// TIA Portal V17 export
// export: Created 2025-03-07T09:16:38.8278492Z, ExportSetting WithDefaults, DisplayName Totally Integrated Automation Portal, DisplayVersion V17 Update 8, DisplayName TIA Portal Openness, DisplayVersion V17 Update 8, DisplayName TIA Portal Version Control Interface, DisplayVersion V17, DisplayName SINAMICS Startdrive Advanced, DisplayVersion V17 SP2, DisplayName SINAMICS Startdrive G110M, G120, G120C, G120D, G120P, G115D, DisplayVersion V17 SP2, DisplayName SINAMICS Startdrive G130, G150, S120, S150, SINAMICS MV, S210, DisplayVersion V17 SP2, DisplayName STEP 7 Professional, DisplayVersion V17 Update 8, DisplayName SINUMERIK ONE STEP 7 Toolbox, DisplayVersion V17 Update 12, DisplayName SINUMERIK 840D sl STEP 7 Toolbox, DisplayVersion V17 Update 12, DisplayName STEP 7 Safety, DisplayVersion V17 Update 6, DisplayName WinCC Advanced, DisplayVersion V17 Update 8
FUNCTION "FC2410_PLC_CNC_SIGNALS" : Void   // FC2410, LAD
TITLE = NCK Inputs
{ S7_Optimized_Access := 'FALSE' }
AUTHOR : ETXETAR
VERSION : 1.0
// stored: AutoNumber false, IsIECCheckEnabled false, SetENOAutomatically false, UDAEnableTagReadback false
   VAR_TEMP
      Error : Bool;   // Error
      ErrorCode : Int;   // ErrorCode
   END_VAR
   VAR CONSTANT
      WRITE : Byte := 16#4;
   END_VAR
BEGIN

REGION Network 1: PLC NC SIGNALS 1-8
   // SIGNAL1 --> SEMIAUTO MODE
   // SIGNAL2 --> DRY CYCLE
   // SIGNAL3 --> RUN OUT
   // SIGNAL4 --> BA3
   // SIGNAL5 --> MANUAL LOAD 
   // SIGNAL6 --> GANTRY ROBOT TEST
   // SIGNAL7 --> ROBOT DRY CYCLE
   // SIGNAL8 --> SPARE
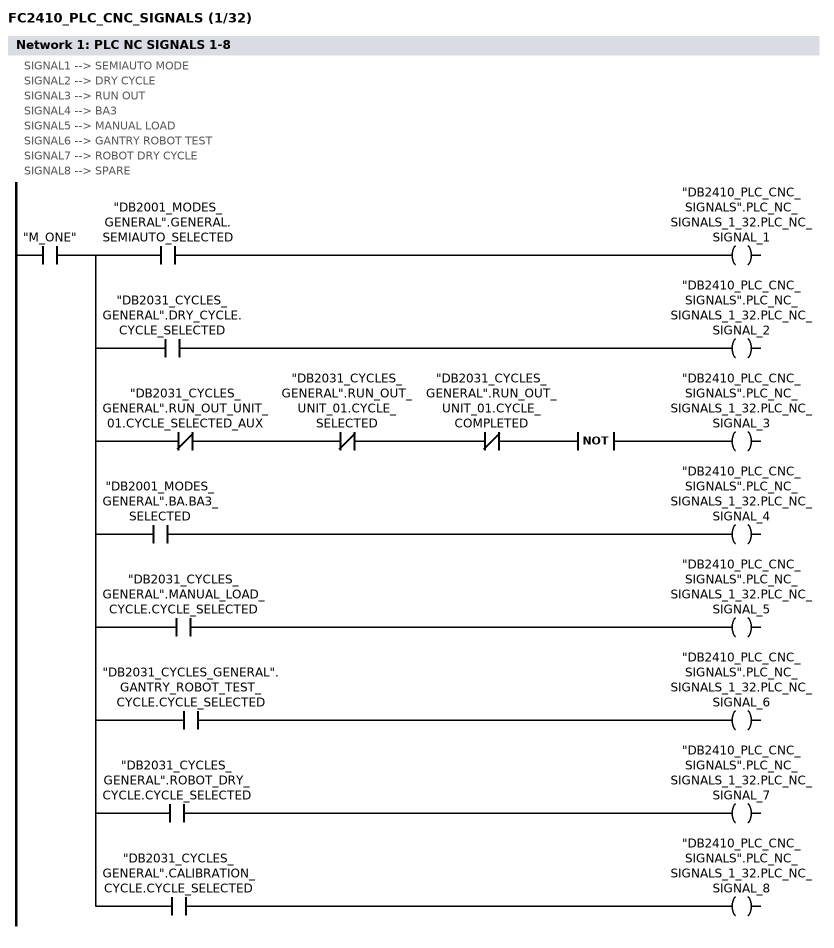
   RUNG wire#powerrail
      Contact( "M_ONE" )
      wire#w1
      Contact( "DB2001_MODES_GENERAL".GENERAL.SEMIAUTO_SELECTED )
      Coil( "DB2410_PLC_CNC_SIGNALS".PLC_NC_SIGNALS_1_32.PLC_NC_SIGNAL_1 )
   END_RUNG
   RUNG wire#w1
      Contact( "DB2031_CYCLES_GENERAL".DRY_CYCLE.CYCLE_SELECTED )
      Coil( "DB2410_PLC_CNC_SIGNALS".PLC_NC_SIGNALS_1_32.PLC_NC_SIGNAL_2 )
   END_RUNG
   RUNG wire#w1
      I_Contact( "DB2031_CYCLES_GENERAL".RUN_OUT_UNIT_01.CYCLE_SELECTED_AUX )
      I_Contact( "DB2031_CYCLES_GENERAL".RUN_OUT_UNIT_01.CYCLE_SELECTED )
      I_Contact( "DB2031_CYCLES_GENERAL".RUN_OUT_UNIT_01.CYCLE_COMPLETED )
      Not()
      Coil( "DB2410_PLC_CNC_SIGNALS".PLC_NC_SIGNALS_1_32.PLC_NC_SIGNAL_3 )
   END_RUNG
   RUNG wire#w1
      Contact( "DB2001_MODES_GENERAL".BA.BA3_SELECTED )
      Coil( "DB2410_PLC_CNC_SIGNALS".PLC_NC_SIGNALS_1_32.PLC_NC_SIGNAL_4 )
   END_RUNG
   RUNG wire#w1
      Contact( "DB2031_CYCLES_GENERAL".MANUAL_LOAD_CYCLE.CYCLE_SELECTED )
      Coil( "DB2410_PLC_CNC_SIGNALS".PLC_NC_SIGNALS_1_32.PLC_NC_SIGNAL_5 )
   END_RUNG
   RUNG wire#w1
      Contact( "DB2031_CYCLES_GENERAL".GANTRY_ROBOT_TEST_CYCLE.CYCLE_SELECTED )
      Coil( "DB2410_PLC_CNC_SIGNALS".PLC_NC_SIGNALS_1_32.PLC_NC_SIGNAL_6 )
   END_RUNG
   RUNG wire#w1
      Contact( "DB2031_CYCLES_GENERAL".ROBOT_DRY_CYCLE.CYCLE_SELECTED )
      Coil( "DB2410_PLC_CNC_SIGNALS".PLC_NC_SIGNALS_1_32.PLC_NC_SIGNAL_7 )
   END_RUNG
   RUNG wire#w1
      Contact( "DB2031_CYCLES_GENERAL".CALIBRATION_CYCLE.CYCLE_SELECTED )
      Coil( "DB2410_PLC_CNC_SIGNALS".PLC_NC_SIGNALS_1_32.PLC_NC_SIGNAL_8 )
   END_RUNG
   // the same network as SCL:
   "DB2410_PLC_CNC_SIGNALS".PLC_NC_SIGNALS_1_32.PLC_NC_SIGNAL_1 := "M_ONE" AND "DB2001_MODES_GENERAL".GENERAL.SEMIAUTO_SELECTED;
   "DB2410_PLC_CNC_SIGNALS".PLC_NC_SIGNALS_1_32.PLC_NC_SIGNAL_2 := "M_ONE" AND "DB2031_CYCLES_GENERAL".DRY_CYCLE.CYCLE_SELECTED;
   "DB2410_PLC_CNC_SIGNALS".PLC_NC_SIGNALS_1_32.PLC_NC_SIGNAL_3 := NOT ("M_ONE" AND NOT "DB2031_CYCLES_GENERAL".RUN_OUT_UNIT_01.CYCLE_SELECTED_AUX AND NOT "DB2031_CYCLES_GENERAL".RUN_OUT_UNIT_01.CYCLE_SELECTED AND NOT "DB2031_CYCLES_GENERAL".RUN_OUT_UNIT_01.CYCLE_COMPLETED);
   "DB2410_PLC_CNC_SIGNALS".PLC_NC_SIGNALS_1_32.PLC_NC_SIGNAL_4 := "M_ONE" AND "DB2001_MODES_GENERAL".BA.BA3_SELECTED;
   "DB2410_PLC_CNC_SIGNALS".PLC_NC_SIGNALS_1_32.PLC_NC_SIGNAL_5 := "M_ONE" AND "DB2031_CYCLES_GENERAL".MANUAL_LOAD_CYCLE.CYCLE_SELECTED;
   "DB2410_PLC_CNC_SIGNALS".PLC_NC_SIGNALS_1_32.PLC_NC_SIGNAL_6 := "M_ONE" AND "DB2031_CYCLES_GENERAL".GANTRY_ROBOT_TEST_CYCLE.CYCLE_SELECTED;
   "DB2410_PLC_CNC_SIGNALS".PLC_NC_SIGNALS_1_32.PLC_NC_SIGNAL_7 := "M_ONE" AND "DB2031_CYCLES_GENERAL".ROBOT_DRY_CYCLE.CYCLE_SELECTED;
   "DB2410_PLC_CNC_SIGNALS".PLC_NC_SIGNALS_1_32.PLC_NC_SIGNAL_8 := "M_ONE" AND "DB2031_CYCLES_GENERAL".CALIBRATION_CYCLE.CYCLE_SELECTED;
END_REGION

REGION Network 2: PLC NC SIGNALS 9-16
   // SIGNAL9 --> SPARE
   // SIGNAL10 --> SPARE
   // SIGNAL11 --> SPARE
   // SIGNAL12 --> SPARE
   // SIGNAL13 --> SPARE
   // SIGNAL14 --> SPARE
   // SIGNAL15 --> SPARE
   // SIGNAL16 --> SPARE
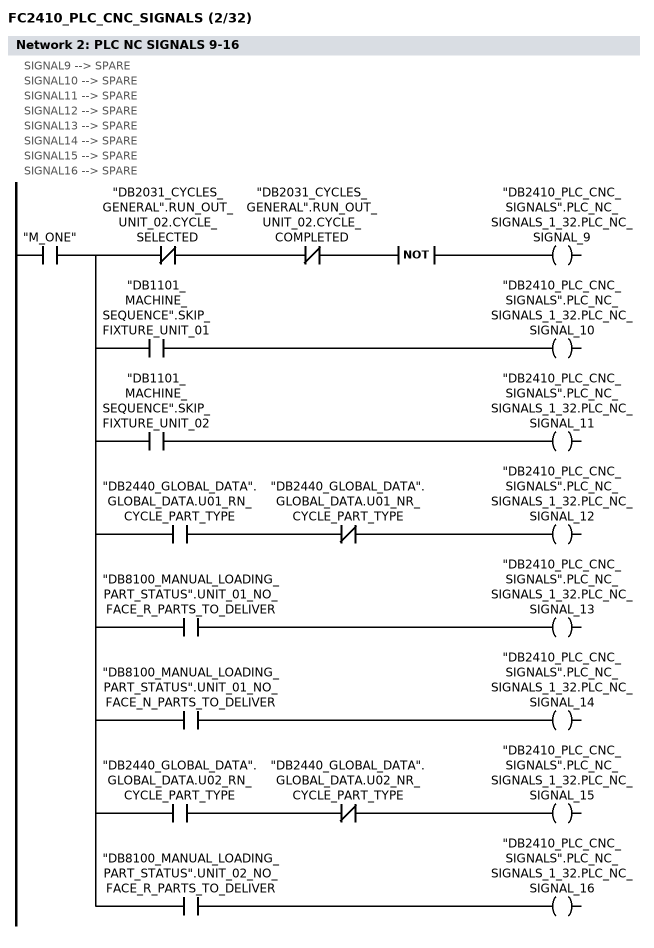
   RUNG wire#powerrail
      Contact( "M_ONE" )
      wire#w1
      I_Contact( "DB2031_CYCLES_GENERAL".RUN_OUT_UNIT_02.CYCLE_SELECTED )
      I_Contact( "DB2031_CYCLES_GENERAL".RUN_OUT_UNIT_02.CYCLE_COMPLETED )
      Not()
      Coil( "DB2410_PLC_CNC_SIGNALS".PLC_NC_SIGNALS_1_32.PLC_NC_SIGNAL_9 )
   END_RUNG
   RUNG wire#w1
      Contact( "DB1101_MACHINE_SEQUENCE".SKIP_FIXTURE_UNIT_01 )
      Coil( "DB2410_PLC_CNC_SIGNALS".PLC_NC_SIGNALS_1_32.PLC_NC_SIGNAL_10 )
   END_RUNG
   RUNG wire#w1
      Contact( "DB1101_MACHINE_SEQUENCE".SKIP_FIXTURE_UNIT_02 )
      Coil( "DB2410_PLC_CNC_SIGNALS".PLC_NC_SIGNALS_1_32.PLC_NC_SIGNAL_11 )
   END_RUNG
   RUNG wire#w1
      Contact( "DB2440_GLOBAL_DATA".GLOBAL_DATA.U01_RN_CYCLE_PART_TYPE )
      I_Contact( "DB2440_GLOBAL_DATA".GLOBAL_DATA.U01_NR_CYCLE_PART_TYPE )
      Coil( "DB2410_PLC_CNC_SIGNALS".PLC_NC_SIGNALS_1_32.PLC_NC_SIGNAL_12 )
   END_RUNG
   RUNG wire#w1
      Contact( "DB8100_MANUAL_LOADING_PART_STATUS".UNIT_01_NO_FACE_R_PARTS_TO_DELIVER )
      Coil( "DB2410_PLC_CNC_SIGNALS".PLC_NC_SIGNALS_1_32.PLC_NC_SIGNAL_13 )
   END_RUNG
   RUNG wire#w1
      Contact( "DB8100_MANUAL_LOADING_PART_STATUS".UNIT_01_NO_FACE_N_PARTS_TO_DELIVER )
      Coil( "DB2410_PLC_CNC_SIGNALS".PLC_NC_SIGNALS_1_32.PLC_NC_SIGNAL_14 )
   END_RUNG
   RUNG wire#w1
      Contact( "DB2440_GLOBAL_DATA".GLOBAL_DATA.U02_RN_CYCLE_PART_TYPE )
      I_Contact( "DB2440_GLOBAL_DATA".GLOBAL_DATA.U02_NR_CYCLE_PART_TYPE )
      Coil( "DB2410_PLC_CNC_SIGNALS".PLC_NC_SIGNALS_1_32.PLC_NC_SIGNAL_15 )
   END_RUNG
   RUNG wire#w1
      Contact( "DB8100_MANUAL_LOADING_PART_STATUS".UNIT_02_NO_FACE_R_PARTS_TO_DELIVER )
      Coil( "DB2410_PLC_CNC_SIGNALS".PLC_NC_SIGNALS_1_32.PLC_NC_SIGNAL_16 )
   END_RUNG
   // the same network as SCL:
   "DB2410_PLC_CNC_SIGNALS".PLC_NC_SIGNALS_1_32.PLC_NC_SIGNAL_9 := NOT ("M_ONE" AND NOT "DB2031_CYCLES_GENERAL".RUN_OUT_UNIT_02.CYCLE_SELECTED AND NOT "DB2031_CYCLES_GENERAL".RUN_OUT_UNIT_02.CYCLE_COMPLETED);
   "DB2410_PLC_CNC_SIGNALS".PLC_NC_SIGNALS_1_32.PLC_NC_SIGNAL_10 := "M_ONE" AND "DB1101_MACHINE_SEQUENCE".SKIP_FIXTURE_UNIT_01;
   "DB2410_PLC_CNC_SIGNALS".PLC_NC_SIGNALS_1_32.PLC_NC_SIGNAL_11 := "M_ONE" AND "DB1101_MACHINE_SEQUENCE".SKIP_FIXTURE_UNIT_02;
   "DB2410_PLC_CNC_SIGNALS".PLC_NC_SIGNALS_1_32.PLC_NC_SIGNAL_12 := "M_ONE" AND "DB2440_GLOBAL_DATA".GLOBAL_DATA.U01_RN_CYCLE_PART_TYPE AND NOT "DB2440_GLOBAL_DATA".GLOBAL_DATA.U01_NR_CYCLE_PART_TYPE;
   "DB2410_PLC_CNC_SIGNALS".PLC_NC_SIGNALS_1_32.PLC_NC_SIGNAL_13 := "M_ONE" AND "DB8100_MANUAL_LOADING_PART_STATUS".UNIT_01_NO_FACE_R_PARTS_TO_DELIVER;
   "DB2410_PLC_CNC_SIGNALS".PLC_NC_SIGNALS_1_32.PLC_NC_SIGNAL_14 := "M_ONE" AND "DB8100_MANUAL_LOADING_PART_STATUS".UNIT_01_NO_FACE_N_PARTS_TO_DELIVER;
   "DB2410_PLC_CNC_SIGNALS".PLC_NC_SIGNALS_1_32.PLC_NC_SIGNAL_15 := "M_ONE" AND "DB2440_GLOBAL_DATA".GLOBAL_DATA.U02_RN_CYCLE_PART_TYPE AND NOT "DB2440_GLOBAL_DATA".GLOBAL_DATA.U02_NR_CYCLE_PART_TYPE;
   "DB2410_PLC_CNC_SIGNALS".PLC_NC_SIGNALS_1_32.PLC_NC_SIGNAL_16 := "M_ONE" AND "DB8100_MANUAL_LOADING_PART_STATUS".UNIT_02_NO_FACE_R_PARTS_TO_DELIVER;
END_REGION

REGION Network 3: PLC NC SIGNALS 17-24
   // SIGNAL17 --> STOP END OF CYCLE
   // SIGNAL18 --> SPARE
   // SIGNAL19 --> SPARE
   // SIGNAL20 --> SPARE
   // SIGNAL21 --> SPARE
   // SIGNAL22 --> SPARE
   // SIGNAL23 --> SPARE
   // SIGNAL24 --> SPARE
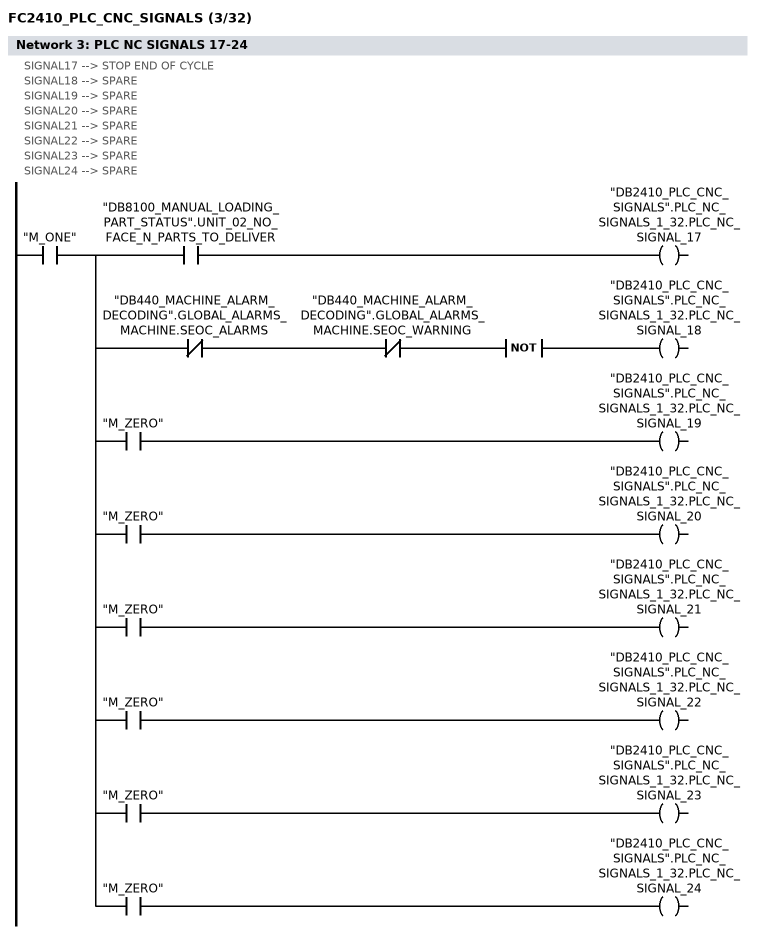
   RUNG wire#powerrail
      Contact( "M_ONE" )
      wire#w1
      Contact( "DB8100_MANUAL_LOADING_PART_STATUS".UNIT_02_NO_FACE_N_PARTS_TO_DELIVER )
      Coil( "DB2410_PLC_CNC_SIGNALS".PLC_NC_SIGNALS_1_32.PLC_NC_SIGNAL_17 )
   END_RUNG
   RUNG wire#w1
      I_Contact( "DB440_MACHINE_ALARM_DECODING".GLOBAL_ALARMS_MACHINE.SEOC_ALARMS )
      I_Contact( "DB440_MACHINE_ALARM_DECODING".GLOBAL_ALARMS_MACHINE.SEOC_WARNING )
      Not()
      Coil( "DB2410_PLC_CNC_SIGNALS".PLC_NC_SIGNALS_1_32.PLC_NC_SIGNAL_18 )
   END_RUNG
   RUNG wire#w1
      Contact( "M_ZERO" )
      Coil( "DB2410_PLC_CNC_SIGNALS".PLC_NC_SIGNALS_1_32.PLC_NC_SIGNAL_19 )
   END_RUNG
   RUNG wire#w1
      Contact( "M_ZERO" )
      Coil( "DB2410_PLC_CNC_SIGNALS".PLC_NC_SIGNALS_1_32.PLC_NC_SIGNAL_20 )
   END_RUNG
   RUNG wire#w1
      Contact( "M_ZERO" )
      Coil( "DB2410_PLC_CNC_SIGNALS".PLC_NC_SIGNALS_1_32.PLC_NC_SIGNAL_21 )
   END_RUNG
   RUNG wire#w1
      Contact( "M_ZERO" )
      Coil( "DB2410_PLC_CNC_SIGNALS".PLC_NC_SIGNALS_1_32.PLC_NC_SIGNAL_22 )
   END_RUNG
   RUNG wire#w1
      Contact( "M_ZERO" )
      Coil( "DB2410_PLC_CNC_SIGNALS".PLC_NC_SIGNALS_1_32.PLC_NC_SIGNAL_23 )
   END_RUNG
   RUNG wire#w1
      Contact( "M_ZERO" )
      Coil( "DB2410_PLC_CNC_SIGNALS".PLC_NC_SIGNALS_1_32.PLC_NC_SIGNAL_24 )
   END_RUNG
   // the same network as SCL:
   "DB2410_PLC_CNC_SIGNALS".PLC_NC_SIGNALS_1_32.PLC_NC_SIGNAL_17 := "M_ONE" AND "DB8100_MANUAL_LOADING_PART_STATUS".UNIT_02_NO_FACE_N_PARTS_TO_DELIVER;
   "DB2410_PLC_CNC_SIGNALS".PLC_NC_SIGNALS_1_32.PLC_NC_SIGNAL_18 := NOT ("M_ONE" AND NOT "DB440_MACHINE_ALARM_DECODING".GLOBAL_ALARMS_MACHINE.SEOC_ALARMS AND NOT "DB440_MACHINE_ALARM_DECODING".GLOBAL_ALARMS_MACHINE.SEOC_WARNING);
   "DB2410_PLC_CNC_SIGNALS".PLC_NC_SIGNALS_1_32.PLC_NC_SIGNAL_19 := "M_ONE" AND "M_ZERO";
   "DB2410_PLC_CNC_SIGNALS".PLC_NC_SIGNALS_1_32.PLC_NC_SIGNAL_20 := "M_ONE" AND "M_ZERO";
   "DB2410_PLC_CNC_SIGNALS".PLC_NC_SIGNALS_1_32.PLC_NC_SIGNAL_21 := "M_ONE" AND "M_ZERO";
   "DB2410_PLC_CNC_SIGNALS".PLC_NC_SIGNALS_1_32.PLC_NC_SIGNAL_22 := "M_ONE" AND "M_ZERO";
   "DB2410_PLC_CNC_SIGNALS".PLC_NC_SIGNALS_1_32.PLC_NC_SIGNAL_23 := "M_ONE" AND "M_ZERO";
   "DB2410_PLC_CNC_SIGNALS".PLC_NC_SIGNALS_1_32.PLC_NC_SIGNAL_24 := "M_ONE" AND "M_ZERO";
END_REGION

REGION Network 4: PLC NC SIGNALS 25-32
   // SIGNAL25 --> CLEAR TO LOAD UNLOAD MACHINE UNIT 01
   // SIGNAL26 --> CLEAR TO LOAD UNLOAD MACHINE UNIT 02
   // SIGNAL27 --> ROBOT OUT OF COLLISION UNIT 01
   // SIGNAL28 --> ROBOT OUT OF COLLISION UNIT 02
   // SIGNAL29 --> SPARE
   // SIGNAL30 --> SPARE
   // SIGNAL31 --> SPARE
   // SIGNAL32 --> SPARE
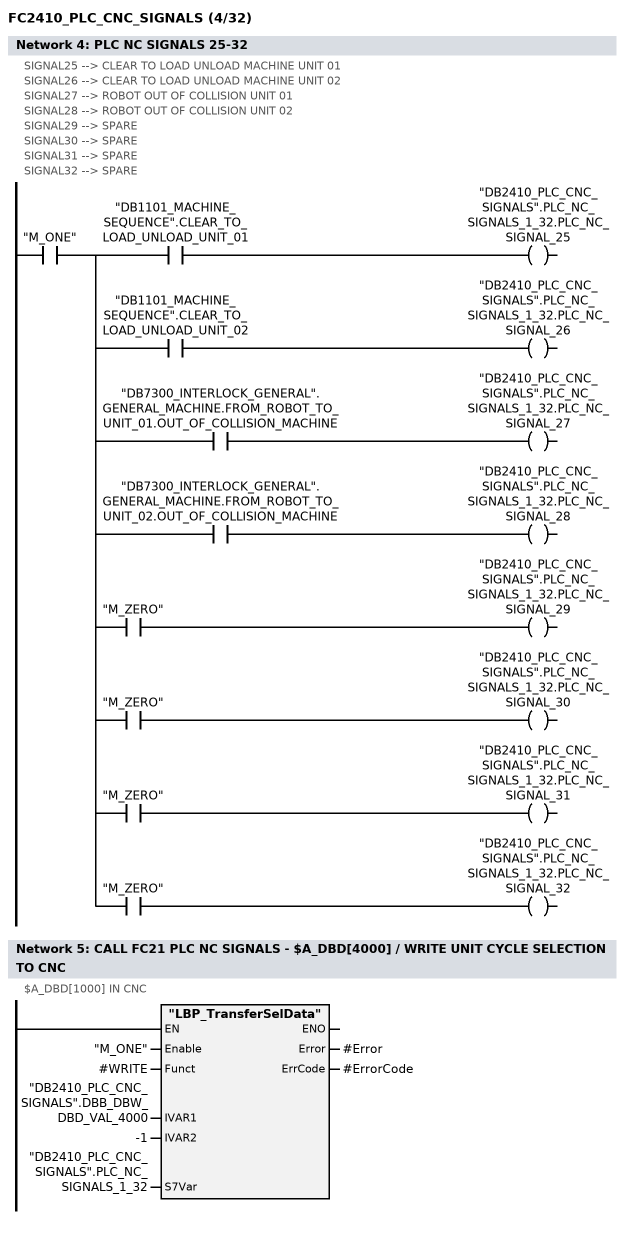
   RUNG wire#powerrail
      Contact( "M_ONE" )
      wire#w1
      Contact( "DB1101_MACHINE_SEQUENCE".CLEAR_TO_LOAD_UNLOAD_UNIT_01 )
      Coil( "DB2410_PLC_CNC_SIGNALS".PLC_NC_SIGNALS_1_32.PLC_NC_SIGNAL_25 )
   END_RUNG
   RUNG wire#w1
      Contact( "DB1101_MACHINE_SEQUENCE".CLEAR_TO_LOAD_UNLOAD_UNIT_02 )
      Coil( "DB2410_PLC_CNC_SIGNALS".PLC_NC_SIGNALS_1_32.PLC_NC_SIGNAL_26 )
   END_RUNG
   RUNG wire#w1
      Contact( "DB7300_INTERLOCK_GENERAL".GENERAL_MACHINE.FROM_ROBOT_TO_UNIT_01.OUT_OF_COLLISION_MACHINE )
      Coil( "DB2410_PLC_CNC_SIGNALS".PLC_NC_SIGNALS_1_32.PLC_NC_SIGNAL_27 )
   END_RUNG
   RUNG wire#w1
      Contact( "DB7300_INTERLOCK_GENERAL".GENERAL_MACHINE.FROM_ROBOT_TO_UNIT_02.OUT_OF_COLLISION_MACHINE )
      Coil( "DB2410_PLC_CNC_SIGNALS".PLC_NC_SIGNALS_1_32.PLC_NC_SIGNAL_28 )
   END_RUNG
   RUNG wire#w1
      Contact( "M_ZERO" )
      Coil( "DB2410_PLC_CNC_SIGNALS".PLC_NC_SIGNALS_1_32.PLC_NC_SIGNAL_29 )
   END_RUNG
   RUNG wire#w1
      Contact( "M_ZERO" )
      Coil( "DB2410_PLC_CNC_SIGNALS".PLC_NC_SIGNALS_1_32.PLC_NC_SIGNAL_30 )
   END_RUNG
   RUNG wire#w1
      Contact( "M_ZERO" )
      Coil( "DB2410_PLC_CNC_SIGNALS".PLC_NC_SIGNALS_1_32.PLC_NC_SIGNAL_31 )
   END_RUNG
   RUNG wire#w1
      Contact( "M_ZERO" )
      Coil( "DB2410_PLC_CNC_SIGNALS".PLC_NC_SIGNALS_1_32.PLC_NC_SIGNAL_32 )
   END_RUNG
   // the same network as SCL:
   "DB2410_PLC_CNC_SIGNALS".PLC_NC_SIGNALS_1_32.PLC_NC_SIGNAL_25 := "M_ONE" AND "DB1101_MACHINE_SEQUENCE".CLEAR_TO_LOAD_UNLOAD_UNIT_01;
   "DB2410_PLC_CNC_SIGNALS".PLC_NC_SIGNALS_1_32.PLC_NC_SIGNAL_26 := "M_ONE" AND "DB1101_MACHINE_SEQUENCE".CLEAR_TO_LOAD_UNLOAD_UNIT_02;
   "DB2410_PLC_CNC_SIGNALS".PLC_NC_SIGNALS_1_32.PLC_NC_SIGNAL_27 := "M_ONE" AND "DB7300_INTERLOCK_GENERAL".GENERAL_MACHINE.FROM_ROBOT_TO_UNIT_01.OUT_OF_COLLISION_MACHINE;
   "DB2410_PLC_CNC_SIGNALS".PLC_NC_SIGNALS_1_32.PLC_NC_SIGNAL_28 := "M_ONE" AND "DB7300_INTERLOCK_GENERAL".GENERAL_MACHINE.FROM_ROBOT_TO_UNIT_02.OUT_OF_COLLISION_MACHINE;
   "DB2410_PLC_CNC_SIGNALS".PLC_NC_SIGNALS_1_32.PLC_NC_SIGNAL_29 := "M_ONE" AND "M_ZERO";
   "DB2410_PLC_CNC_SIGNALS".PLC_NC_SIGNALS_1_32.PLC_NC_SIGNAL_30 := "M_ONE" AND "M_ZERO";
   "DB2410_PLC_CNC_SIGNALS".PLC_NC_SIGNALS_1_32.PLC_NC_SIGNAL_31 := "M_ONE" AND "M_ZERO";
   "DB2410_PLC_CNC_SIGNALS".PLC_NC_SIGNALS_1_32.PLC_NC_SIGNAL_32 := "M_ONE" AND "M_ZERO";
END_REGION

REGION Network 5: CALL FC21 PLC NC SIGNALS - $A_DBD[4000] / WRITE UNIT CYCLE SELECTION TO CNC
   // $A_DBD[1000] IN CNC
   RUNG wire#powerrail
      "LBP_TransferSelData"(Enable := "M_ONE", Funct := #WRITE, IVAR1 := "DB2410_PLC_CNC_SIGNALS".DBB_DBW_DBD_VAL_4000, IVAR2 := -1, S7Var := "DB2410_PLC_CNC_SIGNALS".PLC_NC_SIGNALS_1_32, Error => #Error, ErrCode => #ErrorCode)
   END_RUNG
   // the same network as SCL:
   "LBP_TransferSelData"(Enable := "M_ONE",
                         Funct := #WRITE,
                         IVAR1 := "DB2410_PLC_CNC_SIGNALS".DBB_DBW_DBD_VAL_4000,
                         IVAR2 := -1,
                         S7Var := "DB2410_PLC_CNC_SIGNALS".PLC_NC_SIGNALS_1_32,
                         Error => #Error,
                         ErrCode => #ErrorCode);
END_REGION

REGION Network 6: PLC NC SIGNALS 33-40
   // SIGNAL33 --> TOOL MAZAGINE CHECK HOLDERS 01R
   // SIGNAL34 --> CLEAN TOOL HOLDERS ENABLED 01R
   // SIGNAL35 --> RFID ENABLED 01R
   // SIGNAL36 --> TOOL RFID TAG PRESENT 01R
   // SIGNAL37 --> TOOL CLAMPING DIFFERENCE ALARM 01R
   // SIGNAL38 --> PROBE ENABLED 01R
   // SIGNAL39 --> SPARE
   // SIGNAL40 --> SPARE
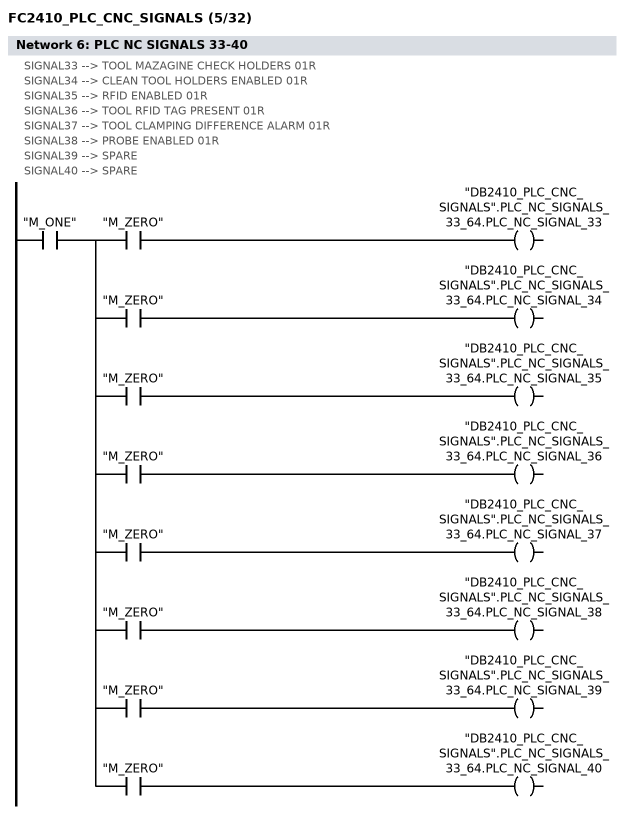
   RUNG wire#powerrail
      Contact( "M_ONE" )
      wire#w1
      Contact( "M_ZERO" )
      Coil( "DB2410_PLC_CNC_SIGNALS".PLC_NC_SIGNALS_33_64.PLC_NC_SIGNAL_33 )
   END_RUNG
   RUNG wire#w1
      Contact( "M_ZERO" )
      Coil( "DB2410_PLC_CNC_SIGNALS".PLC_NC_SIGNALS_33_64.PLC_NC_SIGNAL_34 )
   END_RUNG
   RUNG wire#w1
      Contact( "M_ZERO" )
      Coil( "DB2410_PLC_CNC_SIGNALS".PLC_NC_SIGNALS_33_64.PLC_NC_SIGNAL_35 )
   END_RUNG
   RUNG wire#w1
      Contact( "M_ZERO" )
      Coil( "DB2410_PLC_CNC_SIGNALS".PLC_NC_SIGNALS_33_64.PLC_NC_SIGNAL_36 )
   END_RUNG
   RUNG wire#w1
      Contact( "M_ZERO" )
      Coil( "DB2410_PLC_CNC_SIGNALS".PLC_NC_SIGNALS_33_64.PLC_NC_SIGNAL_37 )
   END_RUNG
   RUNG wire#w1
      Contact( "M_ZERO" )
      Coil( "DB2410_PLC_CNC_SIGNALS".PLC_NC_SIGNALS_33_64.PLC_NC_SIGNAL_38 )
   END_RUNG
   RUNG wire#w1
      Contact( "M_ZERO" )
      Coil( "DB2410_PLC_CNC_SIGNALS".PLC_NC_SIGNALS_33_64.PLC_NC_SIGNAL_39 )
   END_RUNG
   RUNG wire#w1
      Contact( "M_ZERO" )
      Coil( "DB2410_PLC_CNC_SIGNALS".PLC_NC_SIGNALS_33_64.PLC_NC_SIGNAL_40 )
   END_RUNG
   // the same network as SCL:
   "DB2410_PLC_CNC_SIGNALS".PLC_NC_SIGNALS_33_64.PLC_NC_SIGNAL_33 := "M_ONE" AND "M_ZERO";
   "DB2410_PLC_CNC_SIGNALS".PLC_NC_SIGNALS_33_64.PLC_NC_SIGNAL_34 := "M_ONE" AND "M_ZERO";
   "DB2410_PLC_CNC_SIGNALS".PLC_NC_SIGNALS_33_64.PLC_NC_SIGNAL_35 := "M_ONE" AND "M_ZERO";
   "DB2410_PLC_CNC_SIGNALS".PLC_NC_SIGNALS_33_64.PLC_NC_SIGNAL_36 := "M_ONE" AND "M_ZERO";
   "DB2410_PLC_CNC_SIGNALS".PLC_NC_SIGNALS_33_64.PLC_NC_SIGNAL_37 := "M_ONE" AND "M_ZERO";
   "DB2410_PLC_CNC_SIGNALS".PLC_NC_SIGNALS_33_64.PLC_NC_SIGNAL_38 := "M_ONE" AND "M_ZERO";
   "DB2410_PLC_CNC_SIGNALS".PLC_NC_SIGNALS_33_64.PLC_NC_SIGNAL_39 := "M_ONE" AND "M_ZERO";
   "DB2410_PLC_CNC_SIGNALS".PLC_NC_SIGNALS_33_64.PLC_NC_SIGNAL_40 := "M_ONE" AND "M_ZERO";
END_REGION

REGION Network 7: PLC NC SIGNALS 41-48
   // SIGNAL41 --> SPARE
   // SIGNAL42 --> SPARE
   // SIGNAL43 --> SPARE
   // SIGNAL44 --> SPARE
   // SIGNAL45 --> SPARE
   // SIGNAL46 --> SPARE
   // SIGNAL47 --> SPARE
   // SIGNAL48 --> SPARE
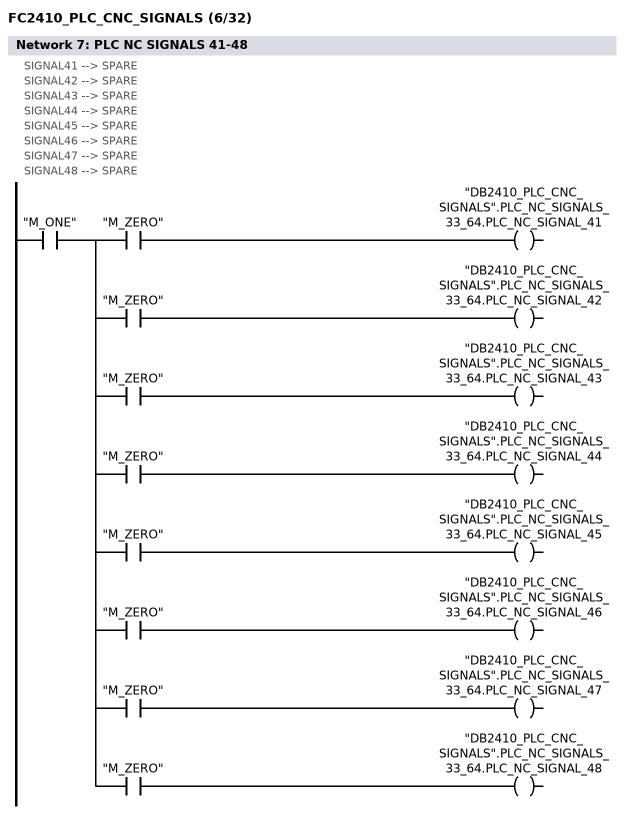
   RUNG wire#powerrail
      Contact( "M_ONE" )
      wire#w1
      Contact( "M_ZERO" )
      Coil( "DB2410_PLC_CNC_SIGNALS".PLC_NC_SIGNALS_33_64.PLC_NC_SIGNAL_41 )
   END_RUNG
   RUNG wire#w1
      Contact( "M_ZERO" )
      Coil( "DB2410_PLC_CNC_SIGNALS".PLC_NC_SIGNALS_33_64.PLC_NC_SIGNAL_42 )
   END_RUNG
   RUNG wire#w1
      Contact( "M_ZERO" )
      Coil( "DB2410_PLC_CNC_SIGNALS".PLC_NC_SIGNALS_33_64.PLC_NC_SIGNAL_43 )
   END_RUNG
   RUNG wire#w1
      Contact( "M_ZERO" )
      Coil( "DB2410_PLC_CNC_SIGNALS".PLC_NC_SIGNALS_33_64.PLC_NC_SIGNAL_44 )
   END_RUNG
   RUNG wire#w1
      Contact( "M_ZERO" )
      Coil( "DB2410_PLC_CNC_SIGNALS".PLC_NC_SIGNALS_33_64.PLC_NC_SIGNAL_45 )
   END_RUNG
   RUNG wire#w1
      Contact( "M_ZERO" )
      Coil( "DB2410_PLC_CNC_SIGNALS".PLC_NC_SIGNALS_33_64.PLC_NC_SIGNAL_46 )
   END_RUNG
   RUNG wire#w1
      Contact( "M_ZERO" )
      Coil( "DB2410_PLC_CNC_SIGNALS".PLC_NC_SIGNALS_33_64.PLC_NC_SIGNAL_47 )
   END_RUNG
   RUNG wire#w1
      Contact( "M_ZERO" )
      Coil( "DB2410_PLC_CNC_SIGNALS".PLC_NC_SIGNALS_33_64.PLC_NC_SIGNAL_48 )
   END_RUNG
   // the same network as SCL:
   "DB2410_PLC_CNC_SIGNALS".PLC_NC_SIGNALS_33_64.PLC_NC_SIGNAL_41 := "M_ONE" AND "M_ZERO";
   "DB2410_PLC_CNC_SIGNALS".PLC_NC_SIGNALS_33_64.PLC_NC_SIGNAL_42 := "M_ONE" AND "M_ZERO";
   "DB2410_PLC_CNC_SIGNALS".PLC_NC_SIGNALS_33_64.PLC_NC_SIGNAL_43 := "M_ONE" AND "M_ZERO";
   "DB2410_PLC_CNC_SIGNALS".PLC_NC_SIGNALS_33_64.PLC_NC_SIGNAL_44 := "M_ONE" AND "M_ZERO";
   "DB2410_PLC_CNC_SIGNALS".PLC_NC_SIGNALS_33_64.PLC_NC_SIGNAL_45 := "M_ONE" AND "M_ZERO";
   "DB2410_PLC_CNC_SIGNALS".PLC_NC_SIGNALS_33_64.PLC_NC_SIGNAL_46 := "M_ONE" AND "M_ZERO";
   "DB2410_PLC_CNC_SIGNALS".PLC_NC_SIGNALS_33_64.PLC_NC_SIGNAL_47 := "M_ONE" AND "M_ZERO";
   "DB2410_PLC_CNC_SIGNALS".PLC_NC_SIGNALS_33_64.PLC_NC_SIGNAL_48 := "M_ONE" AND "M_ZERO";
END_REGION

REGION Network 8: PLC NC SIGNALS 49-56
   // SIGNAL49 --> TOOL MAZAGINE CHECK HOLDERS 01L
   // SIGNAL50 --> CLEAN TOOL HOLDERS ENABLED 01L
   // SIGNAL51 --> RFID ENABLED 01L
   // SIGNAL52 --> TOOL RFID TAG PRESENT 01L
   // SIGNAL53 --> TOOL CLAMPING DIFFERENCE ALARM 01L
   // SIGNAL54 --> PROBE ENABLED 01L
   // SIGNAL55 --> SPARE
   // SIGNAL56 --> SPARE
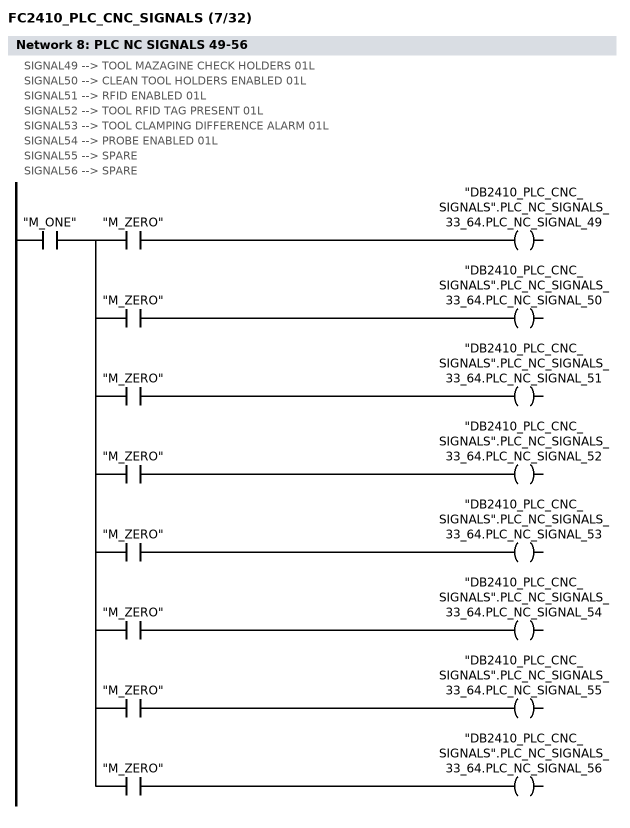
   RUNG wire#powerrail
      Contact( "M_ONE" )
      wire#w1
      Contact( "M_ZERO" )
      Coil( "DB2410_PLC_CNC_SIGNALS".PLC_NC_SIGNALS_33_64.PLC_NC_SIGNAL_49 )
   END_RUNG
   RUNG wire#w1
      Contact( "M_ZERO" )
      Coil( "DB2410_PLC_CNC_SIGNALS".PLC_NC_SIGNALS_33_64.PLC_NC_SIGNAL_50 )
   END_RUNG
   RUNG wire#w1
      Contact( "M_ZERO" )
      Coil( "DB2410_PLC_CNC_SIGNALS".PLC_NC_SIGNALS_33_64.PLC_NC_SIGNAL_51 )
   END_RUNG
   RUNG wire#w1
      Contact( "M_ZERO" )
      Coil( "DB2410_PLC_CNC_SIGNALS".PLC_NC_SIGNALS_33_64.PLC_NC_SIGNAL_52 )
   END_RUNG
   RUNG wire#w1
      Contact( "M_ZERO" )
      Coil( "DB2410_PLC_CNC_SIGNALS".PLC_NC_SIGNALS_33_64.PLC_NC_SIGNAL_53 )
   END_RUNG
   RUNG wire#w1
      Contact( "M_ZERO" )
      Coil( "DB2410_PLC_CNC_SIGNALS".PLC_NC_SIGNALS_33_64.PLC_NC_SIGNAL_54 )
   END_RUNG
   RUNG wire#w1
      Contact( "M_ZERO" )
      Coil( "DB2410_PLC_CNC_SIGNALS".PLC_NC_SIGNALS_33_64.PLC_NC_SIGNAL_55 )
   END_RUNG
   RUNG wire#w1
      Contact( "M_ZERO" )
      Coil( "DB2410_PLC_CNC_SIGNALS".PLC_NC_SIGNALS_33_64.PLC_NC_SIGNAL_56 )
   END_RUNG
   // the same network as SCL:
   "DB2410_PLC_CNC_SIGNALS".PLC_NC_SIGNALS_33_64.PLC_NC_SIGNAL_49 := "M_ONE" AND "M_ZERO";
   "DB2410_PLC_CNC_SIGNALS".PLC_NC_SIGNALS_33_64.PLC_NC_SIGNAL_50 := "M_ONE" AND "M_ZERO";
   "DB2410_PLC_CNC_SIGNALS".PLC_NC_SIGNALS_33_64.PLC_NC_SIGNAL_51 := "M_ONE" AND "M_ZERO";
   "DB2410_PLC_CNC_SIGNALS".PLC_NC_SIGNALS_33_64.PLC_NC_SIGNAL_52 := "M_ONE" AND "M_ZERO";
   "DB2410_PLC_CNC_SIGNALS".PLC_NC_SIGNALS_33_64.PLC_NC_SIGNAL_53 := "M_ONE" AND "M_ZERO";
   "DB2410_PLC_CNC_SIGNALS".PLC_NC_SIGNALS_33_64.PLC_NC_SIGNAL_54 := "M_ONE" AND "M_ZERO";
   "DB2410_PLC_CNC_SIGNALS".PLC_NC_SIGNALS_33_64.PLC_NC_SIGNAL_55 := "M_ONE" AND "M_ZERO";
   "DB2410_PLC_CNC_SIGNALS".PLC_NC_SIGNALS_33_64.PLC_NC_SIGNAL_56 := "M_ONE" AND "M_ZERO";
END_REGION

REGION Network 9: PLC NC SIGNALS 57-64
   // SIGNAL57 --> SPARE
   // SIGNAL58 --> SPARE
   // SIGNAL59 --> SPARE
   // SIGNAL60 --> SPARE
   // SIGNAL61 --> SPARE
   // SIGNAL62 --> SPARE
   // SIGNAL63 --> SPARE
   // SIGNAL64 --> SPARE
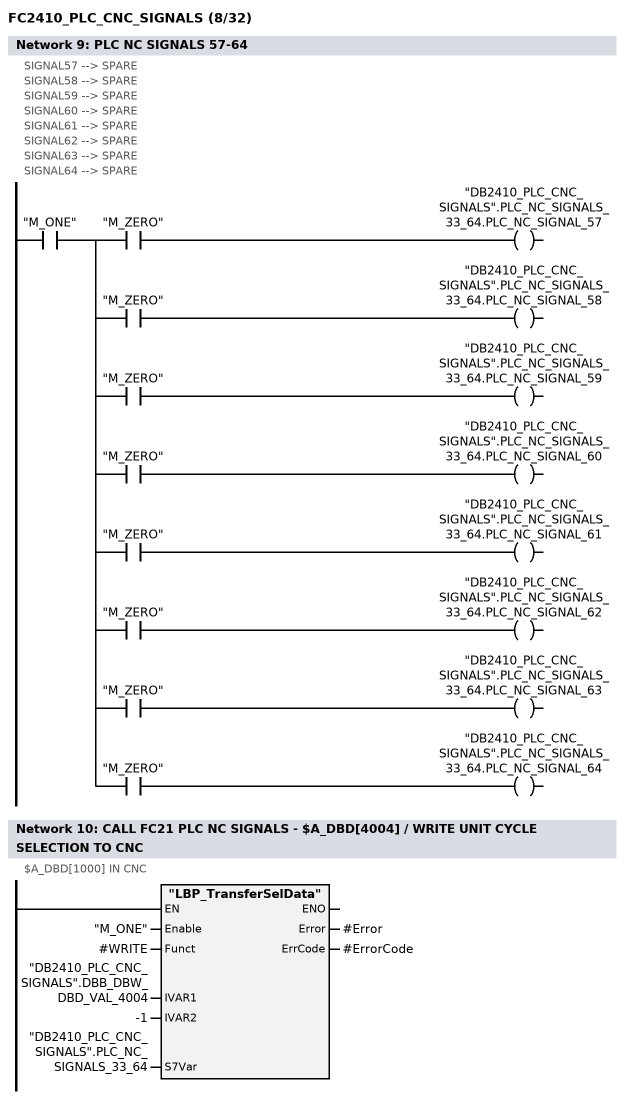
   RUNG wire#powerrail
      Contact( "M_ONE" )
      wire#w1
      Contact( "M_ZERO" )
      Coil( "DB2410_PLC_CNC_SIGNALS".PLC_NC_SIGNALS_33_64.PLC_NC_SIGNAL_57 )
   END_RUNG
   RUNG wire#w1
      Contact( "M_ZERO" )
      Coil( "DB2410_PLC_CNC_SIGNALS".PLC_NC_SIGNALS_33_64.PLC_NC_SIGNAL_58 )
   END_RUNG
   RUNG wire#w1
      Contact( "M_ZERO" )
      Coil( "DB2410_PLC_CNC_SIGNALS".PLC_NC_SIGNALS_33_64.PLC_NC_SIGNAL_59 )
   END_RUNG
   RUNG wire#w1
      Contact( "M_ZERO" )
      Coil( "DB2410_PLC_CNC_SIGNALS".PLC_NC_SIGNALS_33_64.PLC_NC_SIGNAL_60 )
   END_RUNG
   RUNG wire#w1
      Contact( "M_ZERO" )
      Coil( "DB2410_PLC_CNC_SIGNALS".PLC_NC_SIGNALS_33_64.PLC_NC_SIGNAL_61 )
   END_RUNG
   RUNG wire#w1
      Contact( "M_ZERO" )
      Coil( "DB2410_PLC_CNC_SIGNALS".PLC_NC_SIGNALS_33_64.PLC_NC_SIGNAL_62 )
   END_RUNG
   RUNG wire#w1
      Contact( "M_ZERO" )
      Coil( "DB2410_PLC_CNC_SIGNALS".PLC_NC_SIGNALS_33_64.PLC_NC_SIGNAL_63 )
   END_RUNG
   RUNG wire#w1
      Contact( "M_ZERO" )
      Coil( "DB2410_PLC_CNC_SIGNALS".PLC_NC_SIGNALS_33_64.PLC_NC_SIGNAL_64 )
   END_RUNG
   // the same network as SCL:
   "DB2410_PLC_CNC_SIGNALS".PLC_NC_SIGNALS_33_64.PLC_NC_SIGNAL_57 := "M_ONE" AND "M_ZERO";
   "DB2410_PLC_CNC_SIGNALS".PLC_NC_SIGNALS_33_64.PLC_NC_SIGNAL_58 := "M_ONE" AND "M_ZERO";
   "DB2410_PLC_CNC_SIGNALS".PLC_NC_SIGNALS_33_64.PLC_NC_SIGNAL_59 := "M_ONE" AND "M_ZERO";
   "DB2410_PLC_CNC_SIGNALS".PLC_NC_SIGNALS_33_64.PLC_NC_SIGNAL_60 := "M_ONE" AND "M_ZERO";
   "DB2410_PLC_CNC_SIGNALS".PLC_NC_SIGNALS_33_64.PLC_NC_SIGNAL_61 := "M_ONE" AND "M_ZERO";
   "DB2410_PLC_CNC_SIGNALS".PLC_NC_SIGNALS_33_64.PLC_NC_SIGNAL_62 := "M_ONE" AND "M_ZERO";
   "DB2410_PLC_CNC_SIGNALS".PLC_NC_SIGNALS_33_64.PLC_NC_SIGNAL_63 := "M_ONE" AND "M_ZERO";
   "DB2410_PLC_CNC_SIGNALS".PLC_NC_SIGNALS_33_64.PLC_NC_SIGNAL_64 := "M_ONE" AND "M_ZERO";
END_REGION

REGION Network 10: CALL FC21 PLC NC SIGNALS - $A_DBD[4004] / WRITE UNIT CYCLE SELECTION TO CNC
   // $A_DBD[1000] IN CNC
   RUNG wire#powerrail
      "LBP_TransferSelData"(Enable := "M_ONE", Funct := #WRITE, IVAR1 := "DB2410_PLC_CNC_SIGNALS".DBB_DBW_DBD_VAL_4004, IVAR2 := -1, S7Var := "DB2410_PLC_CNC_SIGNALS".PLC_NC_SIGNALS_33_64, Error => #Error, ErrCode => #ErrorCode)
   END_RUNG
   // the same network as SCL:
   "LBP_TransferSelData"(Enable := "M_ONE",
                         Funct := #WRITE,
                         IVAR1 := "DB2410_PLC_CNC_SIGNALS".DBB_DBW_DBD_VAL_4004,
                         IVAR2 := -1,
                         S7Var := "DB2410_PLC_CNC_SIGNALS".PLC_NC_SIGNALS_33_64,
                         Error => #Error,
                         ErrCode => #ErrorCode);
END_REGION

REGION Network 11: PLC NC SIGNALS 65-72
   // SIGNAL65 --> FIXTURE 1 CLAMPED
   // SIGNAL66 --> FIXTURE 1 FULL DEPTHS
   // SIGNAL67 --> FIXTURE 1 WAIT QUALITY CHECK CONFIRMATION
   // SIGNAL68 --> FIXTURE 1 CLAMPED MEMORY
   // SIGNAL69 --> FIXTURE 1 MEASURE CYCLE DONE
   // SIGNAL70 --> SPARE
   // SIGNAL71 --> SPARE
   // SIGNAL72 --> SPARE
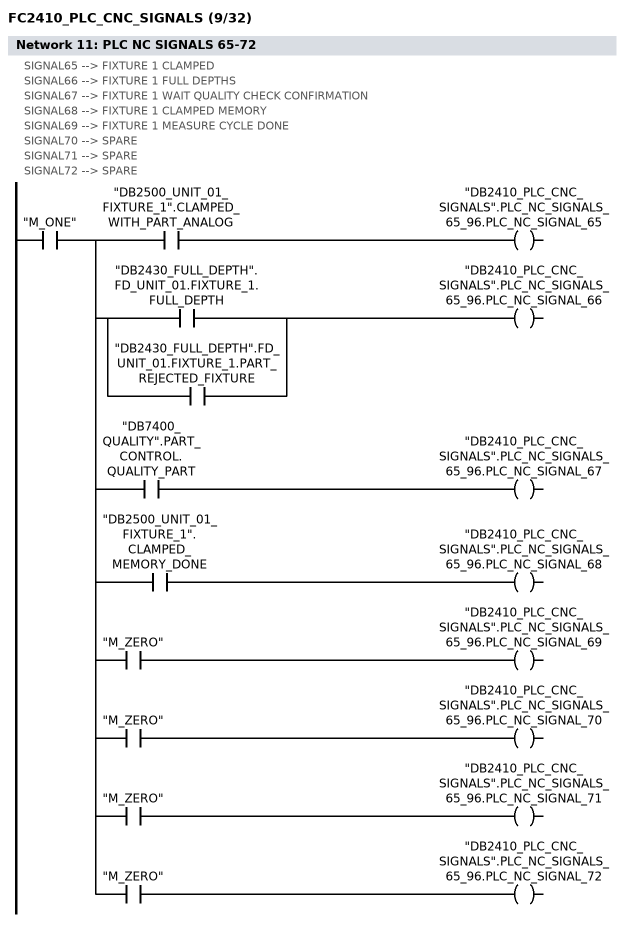
   RUNG wire#powerrail
      Contact( "M_ONE" )
      wire#w1
      Contact( "DB2500_UNIT_01_FIXTURE_1".CLAMPED_WITH_PART_ANALOG )
      Coil( "DB2410_PLC_CNC_SIGNALS".PLC_NC_SIGNALS_65_96.PLC_NC_SIGNAL_65 )
   END_RUNG
   RUNG wire#w1
      Contact( "DB2430_FULL_DEPTH".FD_UNIT_01.FIXTURE_1.FULL_DEPTH )
      wire#w2
      Coil( "DB2410_PLC_CNC_SIGNALS".PLC_NC_SIGNALS_65_96.PLC_NC_SIGNAL_66 )
   END_RUNG
   RUNG wire#w1
      Contact( "DB2430_FULL_DEPTH".FD_UNIT_01.FIXTURE_1.PART_REJECTED_FIXTURE )
   END_RUNG wire#w2
   RUNG wire#w1
      Contact( "DB7400_QUALITY".PART_CONTROL.QUALITY_PART )
      Coil( "DB2410_PLC_CNC_SIGNALS".PLC_NC_SIGNALS_65_96.PLC_NC_SIGNAL_67 )
   END_RUNG
   RUNG wire#w1
      Contact( "DB2500_UNIT_01_FIXTURE_1".CLAMPED_MEMORY_DONE )
      Coil( "DB2410_PLC_CNC_SIGNALS".PLC_NC_SIGNALS_65_96.PLC_NC_SIGNAL_68 )
   END_RUNG
   RUNG wire#w1
      Contact( "M_ZERO" )
      Coil( "DB2410_PLC_CNC_SIGNALS".PLC_NC_SIGNALS_65_96.PLC_NC_SIGNAL_69 )
   END_RUNG
   RUNG wire#w1
      Contact( "M_ZERO" )
      Coil( "DB2410_PLC_CNC_SIGNALS".PLC_NC_SIGNALS_65_96.PLC_NC_SIGNAL_70 )
   END_RUNG
   RUNG wire#w1
      Contact( "M_ZERO" )
      Coil( "DB2410_PLC_CNC_SIGNALS".PLC_NC_SIGNALS_65_96.PLC_NC_SIGNAL_71 )
   END_RUNG
   RUNG wire#w1
      Contact( "M_ZERO" )
      Coil( "DB2410_PLC_CNC_SIGNALS".PLC_NC_SIGNALS_65_96.PLC_NC_SIGNAL_72 )
   END_RUNG
   // the same network as SCL:
   "DB2410_PLC_CNC_SIGNALS".PLC_NC_SIGNALS_65_96.PLC_NC_SIGNAL_65 := "M_ONE" AND "DB2500_UNIT_01_FIXTURE_1".CLAMPED_WITH_PART_ANALOG;
   "DB2410_PLC_CNC_SIGNALS".PLC_NC_SIGNALS_65_96.PLC_NC_SIGNAL_66 := "M_ONE" AND ("DB2430_FULL_DEPTH".FD_UNIT_01.FIXTURE_1.FULL_DEPTH OR "DB2430_FULL_DEPTH".FD_UNIT_01.FIXTURE_1.PART_REJECTED_FIXTURE);
   "DB2410_PLC_CNC_SIGNALS".PLC_NC_SIGNALS_65_96.PLC_NC_SIGNAL_67 := "M_ONE" AND "DB7400_QUALITY".PART_CONTROL.QUALITY_PART;
   "DB2410_PLC_CNC_SIGNALS".PLC_NC_SIGNALS_65_96.PLC_NC_SIGNAL_68 := "M_ONE" AND "DB2500_UNIT_01_FIXTURE_1".CLAMPED_MEMORY_DONE;
   "DB2410_PLC_CNC_SIGNALS".PLC_NC_SIGNALS_65_96.PLC_NC_SIGNAL_69 := "M_ONE" AND "M_ZERO";
   "DB2410_PLC_CNC_SIGNALS".PLC_NC_SIGNALS_65_96.PLC_NC_SIGNAL_70 := "M_ONE" AND "M_ZERO";
   "DB2410_PLC_CNC_SIGNALS".PLC_NC_SIGNALS_65_96.PLC_NC_SIGNAL_71 := "M_ONE" AND "M_ZERO";
   "DB2410_PLC_CNC_SIGNALS".PLC_NC_SIGNALS_65_96.PLC_NC_SIGNAL_72 := "M_ONE" AND "M_ZERO";
END_REGION

REGION Network 12: PLC NC SIGNALS 73-80
   // SIGNAL73 --> FIXTURE 1 PART A PRESENT
   // SIGNAL74 --> FIXTURE 1 PART B PRESENT
   // SIGNAL75 --> FIXTURE 1 PART C PRESENT
   // SIGNAL76 --> FIXTURE 1 PART D PRESENT
   // SIGNAL77 --> SPARE
   // SIGNAL78 --> SPARE
   // SIGNAL79 --> SPARE
   // SIGNAL80 --> SPARE
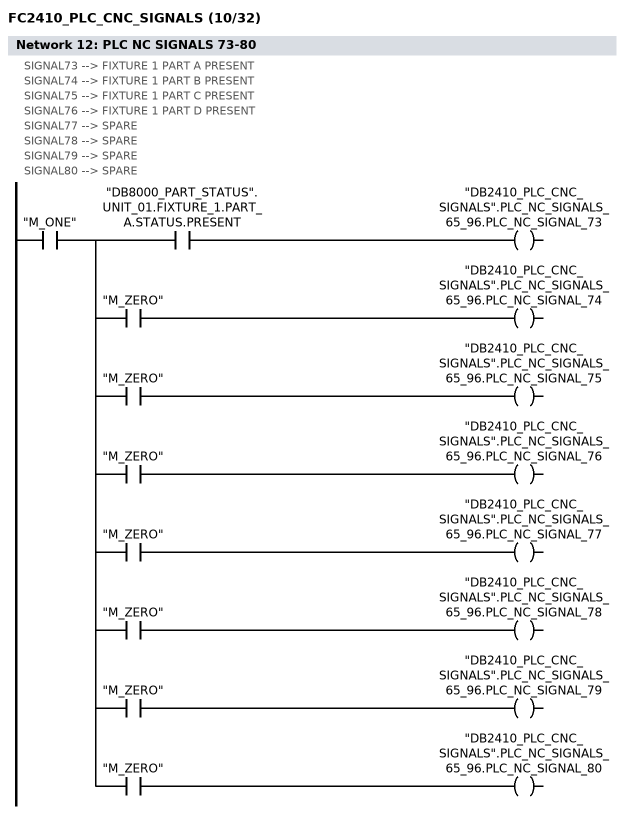
   RUNG wire#powerrail
      Contact( "M_ONE" )
      wire#w1
      Contact( "DB8000_PART_STATUS".UNIT_01.FIXTURE_1.PART_A.STATUS.PRESENT )
      Coil( "DB2410_PLC_CNC_SIGNALS".PLC_NC_SIGNALS_65_96.PLC_NC_SIGNAL_73 )
   END_RUNG
   RUNG wire#w1
      Contact( "M_ZERO" )
      Coil( "DB2410_PLC_CNC_SIGNALS".PLC_NC_SIGNALS_65_96.PLC_NC_SIGNAL_74 )
   END_RUNG
   RUNG wire#w1
      Contact( "M_ZERO" )
      Coil( "DB2410_PLC_CNC_SIGNALS".PLC_NC_SIGNALS_65_96.PLC_NC_SIGNAL_75 )
   END_RUNG
   RUNG wire#w1
      Contact( "M_ZERO" )
      Coil( "DB2410_PLC_CNC_SIGNALS".PLC_NC_SIGNALS_65_96.PLC_NC_SIGNAL_76 )
   END_RUNG
   RUNG wire#w1
      Contact( "M_ZERO" )
      Coil( "DB2410_PLC_CNC_SIGNALS".PLC_NC_SIGNALS_65_96.PLC_NC_SIGNAL_77 )
   END_RUNG
   RUNG wire#w1
      Contact( "M_ZERO" )
      Coil( "DB2410_PLC_CNC_SIGNALS".PLC_NC_SIGNALS_65_96.PLC_NC_SIGNAL_78 )
   END_RUNG
   RUNG wire#w1
      Contact( "M_ZERO" )
      Coil( "DB2410_PLC_CNC_SIGNALS".PLC_NC_SIGNALS_65_96.PLC_NC_SIGNAL_79 )
   END_RUNG
   RUNG wire#w1
      Contact( "M_ZERO" )
      Coil( "DB2410_PLC_CNC_SIGNALS".PLC_NC_SIGNALS_65_96.PLC_NC_SIGNAL_80 )
   END_RUNG
   // the same network as SCL:
   "DB2410_PLC_CNC_SIGNALS".PLC_NC_SIGNALS_65_96.PLC_NC_SIGNAL_73 := "M_ONE" AND "DB8000_PART_STATUS".UNIT_01.FIXTURE_1.PART_A.STATUS.PRESENT;
   "DB2410_PLC_CNC_SIGNALS".PLC_NC_SIGNALS_65_96.PLC_NC_SIGNAL_74 := "M_ONE" AND "M_ZERO";
   "DB2410_PLC_CNC_SIGNALS".PLC_NC_SIGNALS_65_96.PLC_NC_SIGNAL_75 := "M_ONE" AND "M_ZERO";
   "DB2410_PLC_CNC_SIGNALS".PLC_NC_SIGNALS_65_96.PLC_NC_SIGNAL_76 := "M_ONE" AND "M_ZERO";
   "DB2410_PLC_CNC_SIGNALS".PLC_NC_SIGNALS_65_96.PLC_NC_SIGNAL_77 := "M_ONE" AND "M_ZERO";
   "DB2410_PLC_CNC_SIGNALS".PLC_NC_SIGNALS_65_96.PLC_NC_SIGNAL_78 := "M_ONE" AND "M_ZERO";
   "DB2410_PLC_CNC_SIGNALS".PLC_NC_SIGNALS_65_96.PLC_NC_SIGNAL_79 := "M_ONE" AND "M_ZERO";
   "DB2410_PLC_CNC_SIGNALS".PLC_NC_SIGNALS_65_96.PLC_NC_SIGNAL_80 := "M_ONE" AND "M_ZERO";
END_REGION

REGION Network 13: PLC NC SIGNALS 81-88
   // SIGNAL81 --> FIXTURE 1 PART A1 PRESENT
   // SIGNAL82 --> FIXTURE 1 PART B1 PRESENT
   // SIGNAL83 --> FIXTURE 1 PART C1 PRESENT
   // SIGNAL84 --> FIXTURE 1 PART D1 PRESENT
   // SIGNAL85 --> SPARE
   // SIGNAL86 --> SPARE
   // SIGNAL87 --> SPARE
   // SIGNAL88 --> SPARE
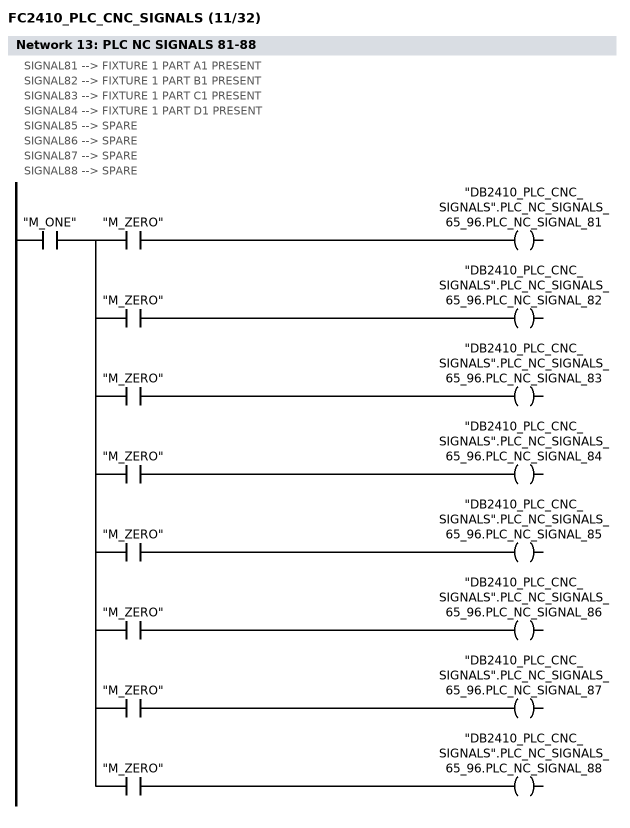
   RUNG wire#powerrail
      Contact( "M_ONE" )
      wire#w1
      Contact( "M_ZERO" )
      Coil( "DB2410_PLC_CNC_SIGNALS".PLC_NC_SIGNALS_65_96.PLC_NC_SIGNAL_81 )
   END_RUNG
   RUNG wire#w1
      Contact( "M_ZERO" )
      Coil( "DB2410_PLC_CNC_SIGNALS".PLC_NC_SIGNALS_65_96.PLC_NC_SIGNAL_82 )
   END_RUNG
   RUNG wire#w1
      Contact( "M_ZERO" )
      Coil( "DB2410_PLC_CNC_SIGNALS".PLC_NC_SIGNALS_65_96.PLC_NC_SIGNAL_83 )
   END_RUNG
   RUNG wire#w1
      Contact( "M_ZERO" )
      Coil( "DB2410_PLC_CNC_SIGNALS".PLC_NC_SIGNALS_65_96.PLC_NC_SIGNAL_84 )
   END_RUNG
   RUNG wire#w1
      Contact( "M_ZERO" )
      Coil( "DB2410_PLC_CNC_SIGNALS".PLC_NC_SIGNALS_65_96.PLC_NC_SIGNAL_85 )
   END_RUNG
   RUNG wire#w1
      Contact( "M_ZERO" )
      Coil( "DB2410_PLC_CNC_SIGNALS".PLC_NC_SIGNALS_65_96.PLC_NC_SIGNAL_86 )
   END_RUNG
   RUNG wire#w1
      Contact( "M_ZERO" )
      Coil( "DB2410_PLC_CNC_SIGNALS".PLC_NC_SIGNALS_65_96.PLC_NC_SIGNAL_87 )
   END_RUNG
   RUNG wire#w1
      Contact( "M_ZERO" )
      Coil( "DB2410_PLC_CNC_SIGNALS".PLC_NC_SIGNALS_65_96.PLC_NC_SIGNAL_88 )
   END_RUNG
   // the same network as SCL:
   "DB2410_PLC_CNC_SIGNALS".PLC_NC_SIGNALS_65_96.PLC_NC_SIGNAL_81 := "M_ONE" AND "M_ZERO";
   "DB2410_PLC_CNC_SIGNALS".PLC_NC_SIGNALS_65_96.PLC_NC_SIGNAL_82 := "M_ONE" AND "M_ZERO";
   "DB2410_PLC_CNC_SIGNALS".PLC_NC_SIGNALS_65_96.PLC_NC_SIGNAL_83 := "M_ONE" AND "M_ZERO";
   "DB2410_PLC_CNC_SIGNALS".PLC_NC_SIGNALS_65_96.PLC_NC_SIGNAL_84 := "M_ONE" AND "M_ZERO";
   "DB2410_PLC_CNC_SIGNALS".PLC_NC_SIGNALS_65_96.PLC_NC_SIGNAL_85 := "M_ONE" AND "M_ZERO";
   "DB2410_PLC_CNC_SIGNALS".PLC_NC_SIGNALS_65_96.PLC_NC_SIGNAL_86 := "M_ONE" AND "M_ZERO";
   "DB2410_PLC_CNC_SIGNALS".PLC_NC_SIGNALS_65_96.PLC_NC_SIGNAL_87 := "M_ONE" AND "M_ZERO";
   "DB2410_PLC_CNC_SIGNALS".PLC_NC_SIGNALS_65_96.PLC_NC_SIGNAL_88 := "M_ONE" AND "M_ZERO";
END_REGION

REGION Network 14: PLC NC SIGNALS 89-96
   // SIGNAL89 --> FIXTURE 1 PART A2 PRESENT
   // SIGNAL90 --> FIXTURE 1 PART B2 PRESENT
   // SIGNAL91 --> FIXTURE 1 PART C2 PRESENT
   // SIGNAL92 --> FIXTURE 1 PART D2 PRESENT
   // SIGNAL93 --> SPARE
   // SIGNAL94 --> SPARE
   // SIGNAL95 --> SPARE
   // SIGNAL96 --> SPARE
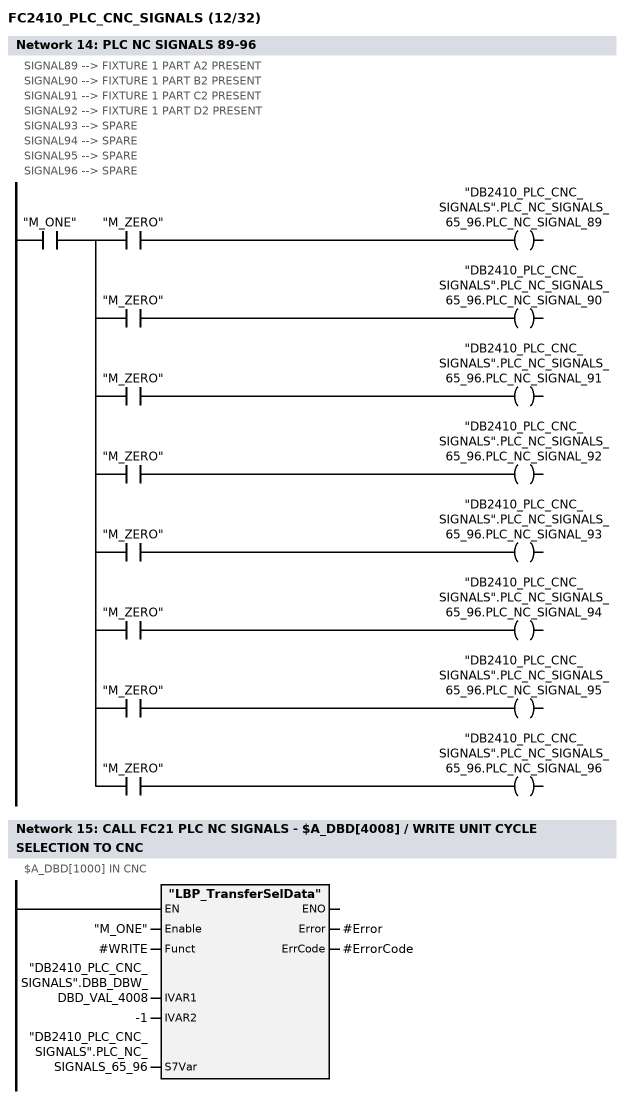
   RUNG wire#powerrail
      Contact( "M_ONE" )
      wire#w1
      Contact( "M_ZERO" )
      Coil( "DB2410_PLC_CNC_SIGNALS".PLC_NC_SIGNALS_65_96.PLC_NC_SIGNAL_89 )
   END_RUNG
   RUNG wire#w1
      Contact( "M_ZERO" )
      Coil( "DB2410_PLC_CNC_SIGNALS".PLC_NC_SIGNALS_65_96.PLC_NC_SIGNAL_90 )
   END_RUNG
   RUNG wire#w1
      Contact( "M_ZERO" )
      Coil( "DB2410_PLC_CNC_SIGNALS".PLC_NC_SIGNALS_65_96.PLC_NC_SIGNAL_91 )
   END_RUNG
   RUNG wire#w1
      Contact( "M_ZERO" )
      Coil( "DB2410_PLC_CNC_SIGNALS".PLC_NC_SIGNALS_65_96.PLC_NC_SIGNAL_92 )
   END_RUNG
   RUNG wire#w1
      Contact( "M_ZERO" )
      Coil( "DB2410_PLC_CNC_SIGNALS".PLC_NC_SIGNALS_65_96.PLC_NC_SIGNAL_93 )
   END_RUNG
   RUNG wire#w1
      Contact( "M_ZERO" )
      Coil( "DB2410_PLC_CNC_SIGNALS".PLC_NC_SIGNALS_65_96.PLC_NC_SIGNAL_94 )
   END_RUNG
   RUNG wire#w1
      Contact( "M_ZERO" )
      Coil( "DB2410_PLC_CNC_SIGNALS".PLC_NC_SIGNALS_65_96.PLC_NC_SIGNAL_95 )
   END_RUNG
   RUNG wire#w1
      Contact( "M_ZERO" )
      Coil( "DB2410_PLC_CNC_SIGNALS".PLC_NC_SIGNALS_65_96.PLC_NC_SIGNAL_96 )
   END_RUNG
   // the same network as SCL:
   "DB2410_PLC_CNC_SIGNALS".PLC_NC_SIGNALS_65_96.PLC_NC_SIGNAL_89 := "M_ONE" AND "M_ZERO";
   "DB2410_PLC_CNC_SIGNALS".PLC_NC_SIGNALS_65_96.PLC_NC_SIGNAL_90 := "M_ONE" AND "M_ZERO";
   "DB2410_PLC_CNC_SIGNALS".PLC_NC_SIGNALS_65_96.PLC_NC_SIGNAL_91 := "M_ONE" AND "M_ZERO";
   "DB2410_PLC_CNC_SIGNALS".PLC_NC_SIGNALS_65_96.PLC_NC_SIGNAL_92 := "M_ONE" AND "M_ZERO";
   "DB2410_PLC_CNC_SIGNALS".PLC_NC_SIGNALS_65_96.PLC_NC_SIGNAL_93 := "M_ONE" AND "M_ZERO";
   "DB2410_PLC_CNC_SIGNALS".PLC_NC_SIGNALS_65_96.PLC_NC_SIGNAL_94 := "M_ONE" AND "M_ZERO";
   "DB2410_PLC_CNC_SIGNALS".PLC_NC_SIGNALS_65_96.PLC_NC_SIGNAL_95 := "M_ONE" AND "M_ZERO";
   "DB2410_PLC_CNC_SIGNALS".PLC_NC_SIGNALS_65_96.PLC_NC_SIGNAL_96 := "M_ONE" AND "M_ZERO";
END_REGION

REGION Network 15: CALL FC21 PLC NC SIGNALS - $A_DBD[4008] / WRITE UNIT CYCLE SELECTION TO CNC
   // $A_DBD[1000] IN CNC
   RUNG wire#powerrail
      "LBP_TransferSelData"(Enable := "M_ONE", Funct := #WRITE, IVAR1 := "DB2410_PLC_CNC_SIGNALS".DBB_DBW_DBD_VAL_4008, IVAR2 := -1, S7Var := "DB2410_PLC_CNC_SIGNALS".PLC_NC_SIGNALS_65_96, Error => #Error, ErrCode => #ErrorCode)
   END_RUNG
   // the same network as SCL:
   "LBP_TransferSelData"(Enable := "M_ONE",
                         Funct := #WRITE,
                         IVAR1 := "DB2410_PLC_CNC_SIGNALS".DBB_DBW_DBD_VAL_4008,
                         IVAR2 := -1,
                         S7Var := "DB2410_PLC_CNC_SIGNALS".PLC_NC_SIGNALS_65_96,
                         Error => #Error,
                         ErrCode => #ErrorCode);
END_REGION

REGION Network 16: PLC NC SIGNALS 97-104
   // SIGNAL97 --> FIXTURE 2 CLAMPED
   // SIGNAL98 --> FIXTURE 2 FULL DEPTHS
   // SIGNAL99 --> FIXTURE 2 WAIT QUALITY CHECK CONFIRMATION
   // SIGNAL100 --> FIXTURE 2 CLAMPED MEMORY
   // SIGNAL101 --> FIXTURE 2 MEASURE CYCLE DONE
   // SIGNAL102 --> SPARE
   // SIGNAL103 --> SPARE
   // SIGNAL104 --> SPARE
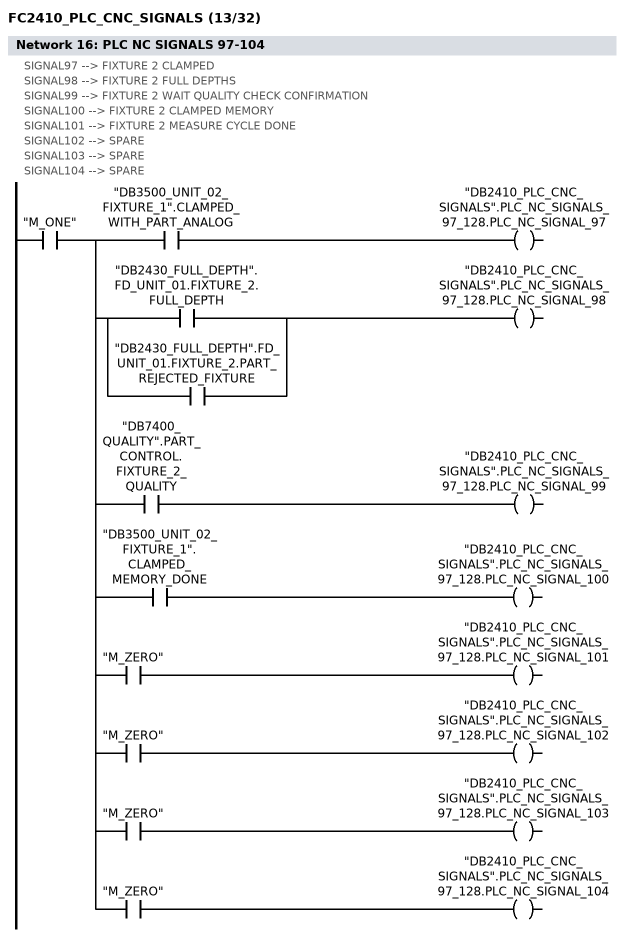
   RUNG wire#powerrail
      Contact( "M_ONE" )
      wire#w1
      Contact( "DB3500_UNIT_02_FIXTURE_1".CLAMPED_WITH_PART_ANALOG )
      Coil( "DB2410_PLC_CNC_SIGNALS".PLC_NC_SIGNALS_97_128.PLC_NC_SIGNAL_97 )
   END_RUNG
   RUNG wire#w1
      Contact( "DB2430_FULL_DEPTH".FD_UNIT_01.FIXTURE_2.FULL_DEPTH )
      wire#w2
      Coil( "DB2410_PLC_CNC_SIGNALS".PLC_NC_SIGNALS_97_128.PLC_NC_SIGNAL_98 )
   END_RUNG
   RUNG wire#w1
      Contact( "DB2430_FULL_DEPTH".FD_UNIT_01.FIXTURE_2.PART_REJECTED_FIXTURE )
   END_RUNG wire#w2
   RUNG wire#w1
      Contact( "DB7400_QUALITY".PART_CONTROL.FIXTURE_2_QUALITY )
      Coil( "DB2410_PLC_CNC_SIGNALS".PLC_NC_SIGNALS_97_128.PLC_NC_SIGNAL_99 )
   END_RUNG
   RUNG wire#w1
      Contact( "DB3500_UNIT_02_FIXTURE_1".CLAMPED_MEMORY_DONE )
      Coil( "DB2410_PLC_CNC_SIGNALS".PLC_NC_SIGNALS_97_128.PLC_NC_SIGNAL_100 )
   END_RUNG
   RUNG wire#w1
      Contact( "M_ZERO" )
      Coil( "DB2410_PLC_CNC_SIGNALS".PLC_NC_SIGNALS_97_128.PLC_NC_SIGNAL_101 )
   END_RUNG
   RUNG wire#w1
      Contact( "M_ZERO" )
      Coil( "DB2410_PLC_CNC_SIGNALS".PLC_NC_SIGNALS_97_128.PLC_NC_SIGNAL_102 )
   END_RUNG
   RUNG wire#w1
      Contact( "M_ZERO" )
      Coil( "DB2410_PLC_CNC_SIGNALS".PLC_NC_SIGNALS_97_128.PLC_NC_SIGNAL_103 )
   END_RUNG
   RUNG wire#w1
      Contact( "M_ZERO" )
      Coil( "DB2410_PLC_CNC_SIGNALS".PLC_NC_SIGNALS_97_128.PLC_NC_SIGNAL_104 )
   END_RUNG
   // the same network as SCL:
   "DB2410_PLC_CNC_SIGNALS".PLC_NC_SIGNALS_97_128.PLC_NC_SIGNAL_97 := "M_ONE" AND "DB3500_UNIT_02_FIXTURE_1".CLAMPED_WITH_PART_ANALOG;
   "DB2410_PLC_CNC_SIGNALS".PLC_NC_SIGNALS_97_128.PLC_NC_SIGNAL_98 := "M_ONE" AND ("DB2430_FULL_DEPTH".FD_UNIT_01.FIXTURE_2.FULL_DEPTH OR "DB2430_FULL_DEPTH".FD_UNIT_01.FIXTURE_2.PART_REJECTED_FIXTURE);
   "DB2410_PLC_CNC_SIGNALS".PLC_NC_SIGNALS_97_128.PLC_NC_SIGNAL_99 := "M_ONE" AND "DB7400_QUALITY".PART_CONTROL.FIXTURE_2_QUALITY;
   "DB2410_PLC_CNC_SIGNALS".PLC_NC_SIGNALS_97_128.PLC_NC_SIGNAL_100 := "M_ONE" AND "DB3500_UNIT_02_FIXTURE_1".CLAMPED_MEMORY_DONE;
   "DB2410_PLC_CNC_SIGNALS".PLC_NC_SIGNALS_97_128.PLC_NC_SIGNAL_101 := "M_ONE" AND "M_ZERO";
   "DB2410_PLC_CNC_SIGNALS".PLC_NC_SIGNALS_97_128.PLC_NC_SIGNAL_102 := "M_ONE" AND "M_ZERO";
   "DB2410_PLC_CNC_SIGNALS".PLC_NC_SIGNALS_97_128.PLC_NC_SIGNAL_103 := "M_ONE" AND "M_ZERO";
   "DB2410_PLC_CNC_SIGNALS".PLC_NC_SIGNALS_97_128.PLC_NC_SIGNAL_104 := "M_ONE" AND "M_ZERO";
END_REGION

REGION Network 17: PLC NC SIGNALS 105-112
   // SIGNAL105 --> FIXTURE 2 PART A PRESENT
   // SIGNAL106 --> FIXTURE 2 PART B PRESENT
   // SIGNAL107 --> FIXTURE 2 PART C PRESENT
   // SIGNAL108 --> FIXTURE 2 PART D PRESENT
   // SIGNAL109 --> SPARE
   // SIGNAL110 --> SPARE
   // SIGNAL111 --> SPARE
   // SIGNAL112 --> SPARE
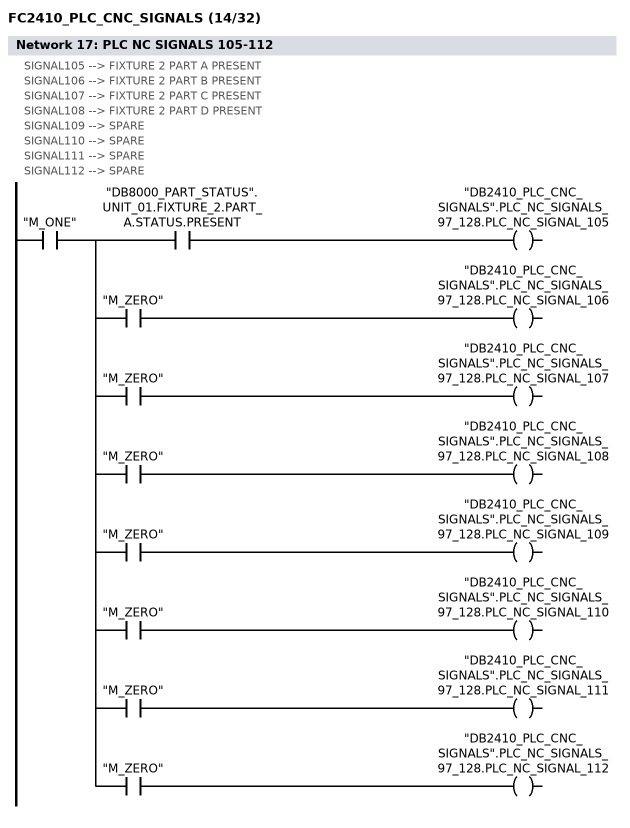
   RUNG wire#powerrail
      Contact( "M_ONE" )
      wire#w1
      Contact( "DB8000_PART_STATUS".UNIT_01.FIXTURE_2.PART_A.STATUS.PRESENT )
      Coil( "DB2410_PLC_CNC_SIGNALS".PLC_NC_SIGNALS_97_128.PLC_NC_SIGNAL_105 )
   END_RUNG
   RUNG wire#w1
      Contact( "M_ZERO" )
      Coil( "DB2410_PLC_CNC_SIGNALS".PLC_NC_SIGNALS_97_128.PLC_NC_SIGNAL_106 )
   END_RUNG
   RUNG wire#w1
      Contact( "M_ZERO" )
      Coil( "DB2410_PLC_CNC_SIGNALS".PLC_NC_SIGNALS_97_128.PLC_NC_SIGNAL_107 )
   END_RUNG
   RUNG wire#w1
      Contact( "M_ZERO" )
      Coil( "DB2410_PLC_CNC_SIGNALS".PLC_NC_SIGNALS_97_128.PLC_NC_SIGNAL_108 )
   END_RUNG
   RUNG wire#w1
      Contact( "M_ZERO" )
      Coil( "DB2410_PLC_CNC_SIGNALS".PLC_NC_SIGNALS_97_128.PLC_NC_SIGNAL_109 )
   END_RUNG
   RUNG wire#w1
      Contact( "M_ZERO" )
      Coil( "DB2410_PLC_CNC_SIGNALS".PLC_NC_SIGNALS_97_128.PLC_NC_SIGNAL_110 )
   END_RUNG
   RUNG wire#w1
      Contact( "M_ZERO" )
      Coil( "DB2410_PLC_CNC_SIGNALS".PLC_NC_SIGNALS_97_128.PLC_NC_SIGNAL_111 )
   END_RUNG
   RUNG wire#w1
      Contact( "M_ZERO" )
      Coil( "DB2410_PLC_CNC_SIGNALS".PLC_NC_SIGNALS_97_128.PLC_NC_SIGNAL_112 )
   END_RUNG
   // the same network as SCL:
   "DB2410_PLC_CNC_SIGNALS".PLC_NC_SIGNALS_97_128.PLC_NC_SIGNAL_105 := "M_ONE" AND "DB8000_PART_STATUS".UNIT_01.FIXTURE_2.PART_A.STATUS.PRESENT;
   "DB2410_PLC_CNC_SIGNALS".PLC_NC_SIGNALS_97_128.PLC_NC_SIGNAL_106 := "M_ONE" AND "M_ZERO";
   "DB2410_PLC_CNC_SIGNALS".PLC_NC_SIGNALS_97_128.PLC_NC_SIGNAL_107 := "M_ONE" AND "M_ZERO";
   "DB2410_PLC_CNC_SIGNALS".PLC_NC_SIGNALS_97_128.PLC_NC_SIGNAL_108 := "M_ONE" AND "M_ZERO";
   "DB2410_PLC_CNC_SIGNALS".PLC_NC_SIGNALS_97_128.PLC_NC_SIGNAL_109 := "M_ONE" AND "M_ZERO";
   "DB2410_PLC_CNC_SIGNALS".PLC_NC_SIGNALS_97_128.PLC_NC_SIGNAL_110 := "M_ONE" AND "M_ZERO";
   "DB2410_PLC_CNC_SIGNALS".PLC_NC_SIGNALS_97_128.PLC_NC_SIGNAL_111 := "M_ONE" AND "M_ZERO";
   "DB2410_PLC_CNC_SIGNALS".PLC_NC_SIGNALS_97_128.PLC_NC_SIGNAL_112 := "M_ONE" AND "M_ZERO";
END_REGION

REGION Network 18: PLC NC SIGNALS 113-120
   // SIGNAL113 --> FIXTURE 2 PART A1 PRESENT
   // SIGNAL114 --> FIXTURE 2 PART B1 PRESENT
   // SIGNAL115 --> FIXTURE 2 PART C1 PRESENT
   // SIGNAL116 --> FIXTURE 2 PART D1 PRESENT
   // SIGNAL117 --> SPARE
   // SIGNAL118 --> SPARE
   // SIGNAL119 --> SPARE
   // SIGNAL120 --> SPARE
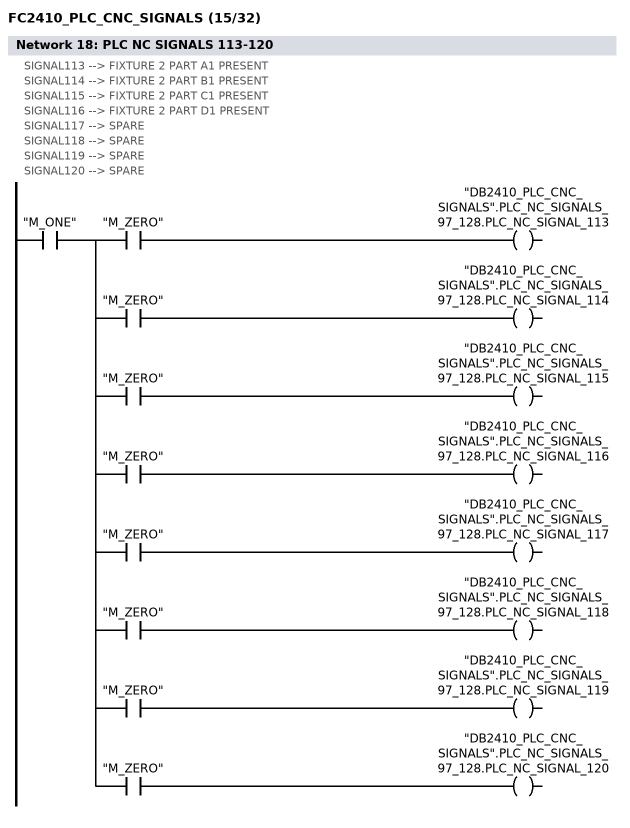
   RUNG wire#powerrail
      Contact( "M_ONE" )
      wire#w1
      Contact( "M_ZERO" )
      Coil( "DB2410_PLC_CNC_SIGNALS".PLC_NC_SIGNALS_97_128.PLC_NC_SIGNAL_113 )
   END_RUNG
   RUNG wire#w1
      Contact( "M_ZERO" )
      Coil( "DB2410_PLC_CNC_SIGNALS".PLC_NC_SIGNALS_97_128.PLC_NC_SIGNAL_114 )
   END_RUNG
   RUNG wire#w1
      Contact( "M_ZERO" )
      Coil( "DB2410_PLC_CNC_SIGNALS".PLC_NC_SIGNALS_97_128.PLC_NC_SIGNAL_115 )
   END_RUNG
   RUNG wire#w1
      Contact( "M_ZERO" )
      Coil( "DB2410_PLC_CNC_SIGNALS".PLC_NC_SIGNALS_97_128.PLC_NC_SIGNAL_116 )
   END_RUNG
   RUNG wire#w1
      Contact( "M_ZERO" )
      Coil( "DB2410_PLC_CNC_SIGNALS".PLC_NC_SIGNALS_97_128.PLC_NC_SIGNAL_117 )
   END_RUNG
   RUNG wire#w1
      Contact( "M_ZERO" )
      Coil( "DB2410_PLC_CNC_SIGNALS".PLC_NC_SIGNALS_97_128.PLC_NC_SIGNAL_118 )
   END_RUNG
   RUNG wire#w1
      Contact( "M_ZERO" )
      Coil( "DB2410_PLC_CNC_SIGNALS".PLC_NC_SIGNALS_97_128.PLC_NC_SIGNAL_119 )
   END_RUNG
   RUNG wire#w1
      Contact( "M_ZERO" )
      Coil( "DB2410_PLC_CNC_SIGNALS".PLC_NC_SIGNALS_97_128.PLC_NC_SIGNAL_120 )
   END_RUNG
   // the same network as SCL:
   "DB2410_PLC_CNC_SIGNALS".PLC_NC_SIGNALS_97_128.PLC_NC_SIGNAL_113 := "M_ONE" AND "M_ZERO";
   "DB2410_PLC_CNC_SIGNALS".PLC_NC_SIGNALS_97_128.PLC_NC_SIGNAL_114 := "M_ONE" AND "M_ZERO";
   "DB2410_PLC_CNC_SIGNALS".PLC_NC_SIGNALS_97_128.PLC_NC_SIGNAL_115 := "M_ONE" AND "M_ZERO";
   "DB2410_PLC_CNC_SIGNALS".PLC_NC_SIGNALS_97_128.PLC_NC_SIGNAL_116 := "M_ONE" AND "M_ZERO";
   "DB2410_PLC_CNC_SIGNALS".PLC_NC_SIGNALS_97_128.PLC_NC_SIGNAL_117 := "M_ONE" AND "M_ZERO";
   "DB2410_PLC_CNC_SIGNALS".PLC_NC_SIGNALS_97_128.PLC_NC_SIGNAL_118 := "M_ONE" AND "M_ZERO";
   "DB2410_PLC_CNC_SIGNALS".PLC_NC_SIGNALS_97_128.PLC_NC_SIGNAL_119 := "M_ONE" AND "M_ZERO";
   "DB2410_PLC_CNC_SIGNALS".PLC_NC_SIGNALS_97_128.PLC_NC_SIGNAL_120 := "M_ONE" AND "M_ZERO";
END_REGION

REGION Network 19: PLC NC SIGNALS 121-128
   // SIGNAL121 --> FIXTURE 2 PART A2 PRESENT
   // SIGNAL122 --> FIXTURE 2 PART B2 PRESENT
   // SIGNAL123 --> FIXTURE 2 PART C2 PRESENT
   // SIGNAL124 --> FIXTURE 2 PART D2 PRESENT
   // SIGNAL125 --> SPARE
   // SIGNAL126 --> SPARE
   // SIGNAL127 --> SPARE
   // SIGNAL128 --> SPARE
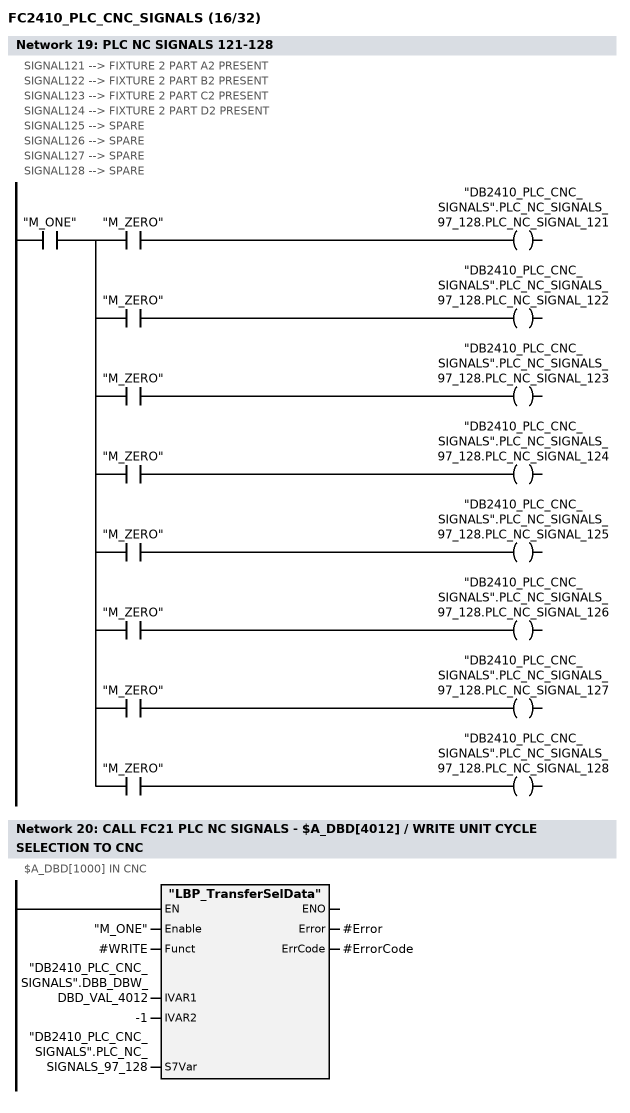
   RUNG wire#powerrail
      Contact( "M_ONE" )
      wire#w1
      Contact( "M_ZERO" )
      Coil( "DB2410_PLC_CNC_SIGNALS".PLC_NC_SIGNALS_97_128.PLC_NC_SIGNAL_121 )
   END_RUNG
   RUNG wire#w1
      Contact( "M_ZERO" )
      Coil( "DB2410_PLC_CNC_SIGNALS".PLC_NC_SIGNALS_97_128.PLC_NC_SIGNAL_122 )
   END_RUNG
   RUNG wire#w1
      Contact( "M_ZERO" )
      Coil( "DB2410_PLC_CNC_SIGNALS".PLC_NC_SIGNALS_97_128.PLC_NC_SIGNAL_123 )
   END_RUNG
   RUNG wire#w1
      Contact( "M_ZERO" )
      Coil( "DB2410_PLC_CNC_SIGNALS".PLC_NC_SIGNALS_97_128.PLC_NC_SIGNAL_124 )
   END_RUNG
   RUNG wire#w1
      Contact( "M_ZERO" )
      Coil( "DB2410_PLC_CNC_SIGNALS".PLC_NC_SIGNALS_97_128.PLC_NC_SIGNAL_125 )
   END_RUNG
   RUNG wire#w1
      Contact( "M_ZERO" )
      Coil( "DB2410_PLC_CNC_SIGNALS".PLC_NC_SIGNALS_97_128.PLC_NC_SIGNAL_126 )
   END_RUNG
   RUNG wire#w1
      Contact( "M_ZERO" )
      Coil( "DB2410_PLC_CNC_SIGNALS".PLC_NC_SIGNALS_97_128.PLC_NC_SIGNAL_127 )
   END_RUNG
   RUNG wire#w1
      Contact( "M_ZERO" )
      Coil( "DB2410_PLC_CNC_SIGNALS".PLC_NC_SIGNALS_97_128.PLC_NC_SIGNAL_128 )
   END_RUNG
   // the same network as SCL:
   "DB2410_PLC_CNC_SIGNALS".PLC_NC_SIGNALS_97_128.PLC_NC_SIGNAL_121 := "M_ONE" AND "M_ZERO";
   "DB2410_PLC_CNC_SIGNALS".PLC_NC_SIGNALS_97_128.PLC_NC_SIGNAL_122 := "M_ONE" AND "M_ZERO";
   "DB2410_PLC_CNC_SIGNALS".PLC_NC_SIGNALS_97_128.PLC_NC_SIGNAL_123 := "M_ONE" AND "M_ZERO";
   "DB2410_PLC_CNC_SIGNALS".PLC_NC_SIGNALS_97_128.PLC_NC_SIGNAL_124 := "M_ONE" AND "M_ZERO";
   "DB2410_PLC_CNC_SIGNALS".PLC_NC_SIGNALS_97_128.PLC_NC_SIGNAL_125 := "M_ONE" AND "M_ZERO";
   "DB2410_PLC_CNC_SIGNALS".PLC_NC_SIGNALS_97_128.PLC_NC_SIGNAL_126 := "M_ONE" AND "M_ZERO";
   "DB2410_PLC_CNC_SIGNALS".PLC_NC_SIGNALS_97_128.PLC_NC_SIGNAL_127 := "M_ONE" AND "M_ZERO";
   "DB2410_PLC_CNC_SIGNALS".PLC_NC_SIGNALS_97_128.PLC_NC_SIGNAL_128 := "M_ONE" AND "M_ZERO";
END_REGION

REGION Network 20: CALL FC21 PLC NC SIGNALS - $A_DBD[4012] / WRITE UNIT CYCLE SELECTION TO CNC
   // $A_DBD[1000] IN CNC
   RUNG wire#powerrail
      "LBP_TransferSelData"(Enable := "M_ONE", Funct := #WRITE, IVAR1 := "DB2410_PLC_CNC_SIGNALS".DBB_DBW_DBD_VAL_4012, IVAR2 := -1, S7Var := "DB2410_PLC_CNC_SIGNALS".PLC_NC_SIGNALS_97_128, Error => #Error, ErrCode => #ErrorCode)
   END_RUNG
   // the same network as SCL:
   "LBP_TransferSelData"(Enable := "M_ONE",
                         Funct := #WRITE,
                         IVAR1 := "DB2410_PLC_CNC_SIGNALS".DBB_DBW_DBD_VAL_4012,
                         IVAR2 := -1,
                         S7Var := "DB2410_PLC_CNC_SIGNALS".PLC_NC_SIGNALS_97_128,
                         Error => #Error,
                         ErrCode => #ErrorCode);
END_REGION

REGION Network 21: PLC NC SIGNALS 129-136
   // SIGNAL129 --> SPARE
   // SIGNAL130 --> SPARE
   // SIGNAL131 --> SPARE
   // SIGNAL132 --> SPARE
   // SIGNAL133 --> SPARE
   // SIGNAL134 --> SPARE
   // SIGNAL135 --> SPARE
   // SIGNAL136 --> SPARE
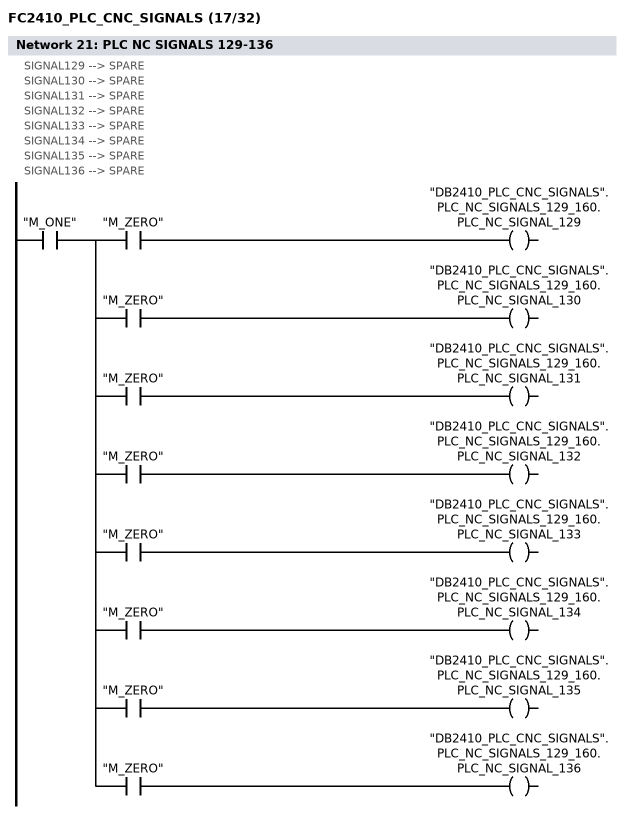
   RUNG wire#powerrail
      Contact( "M_ONE" )
      wire#w1
      Contact( "M_ZERO" )
      Coil( "DB2410_PLC_CNC_SIGNALS".PLC_NC_SIGNALS_129_160.PLC_NC_SIGNAL_129 )
   END_RUNG
   RUNG wire#w1
      Contact( "M_ZERO" )
      Coil( "DB2410_PLC_CNC_SIGNALS".PLC_NC_SIGNALS_129_160.PLC_NC_SIGNAL_130 )
   END_RUNG
   RUNG wire#w1
      Contact( "M_ZERO" )
      Coil( "DB2410_PLC_CNC_SIGNALS".PLC_NC_SIGNALS_129_160.PLC_NC_SIGNAL_131 )
   END_RUNG
   RUNG wire#w1
      Contact( "M_ZERO" )
      Coil( "DB2410_PLC_CNC_SIGNALS".PLC_NC_SIGNALS_129_160.PLC_NC_SIGNAL_132 )
   END_RUNG
   RUNG wire#w1
      Contact( "M_ZERO" )
      Coil( "DB2410_PLC_CNC_SIGNALS".PLC_NC_SIGNALS_129_160.PLC_NC_SIGNAL_133 )
   END_RUNG
   RUNG wire#w1
      Contact( "M_ZERO" )
      Coil( "DB2410_PLC_CNC_SIGNALS".PLC_NC_SIGNALS_129_160.PLC_NC_SIGNAL_134 )
   END_RUNG
   RUNG wire#w1
      Contact( "M_ZERO" )
      Coil( "DB2410_PLC_CNC_SIGNALS".PLC_NC_SIGNALS_129_160.PLC_NC_SIGNAL_135 )
   END_RUNG
   RUNG wire#w1
      Contact( "M_ZERO" )
      Coil( "DB2410_PLC_CNC_SIGNALS".PLC_NC_SIGNALS_129_160.PLC_NC_SIGNAL_136 )
   END_RUNG
   // the same network as SCL:
   "DB2410_PLC_CNC_SIGNALS".PLC_NC_SIGNALS_129_160.PLC_NC_SIGNAL_129 := "M_ONE" AND "M_ZERO";
   "DB2410_PLC_CNC_SIGNALS".PLC_NC_SIGNALS_129_160.PLC_NC_SIGNAL_130 := "M_ONE" AND "M_ZERO";
   "DB2410_PLC_CNC_SIGNALS".PLC_NC_SIGNALS_129_160.PLC_NC_SIGNAL_131 := "M_ONE" AND "M_ZERO";
   "DB2410_PLC_CNC_SIGNALS".PLC_NC_SIGNALS_129_160.PLC_NC_SIGNAL_132 := "M_ONE" AND "M_ZERO";
   "DB2410_PLC_CNC_SIGNALS".PLC_NC_SIGNALS_129_160.PLC_NC_SIGNAL_133 := "M_ONE" AND "M_ZERO";
   "DB2410_PLC_CNC_SIGNALS".PLC_NC_SIGNALS_129_160.PLC_NC_SIGNAL_134 := "M_ONE" AND "M_ZERO";
   "DB2410_PLC_CNC_SIGNALS".PLC_NC_SIGNALS_129_160.PLC_NC_SIGNAL_135 := "M_ONE" AND "M_ZERO";
   "DB2410_PLC_CNC_SIGNALS".PLC_NC_SIGNALS_129_160.PLC_NC_SIGNAL_136 := "M_ONE" AND "M_ZERO";
END_REGION

REGION Network 22: PLC NC SIGNALS 137-144
   // SIGNAL137 --> SPARE
   // SIGNAL138 --> SPARE
   // SIGNAL139 --> SPARE
   // SIGNAL140 --> SPARE
   // SIGNAL141 --> SPARE
   // SIGNAL142 --> SPARE
   // SIGNAL143 --> SPARE
   // SIGNAL144 --> SPARE
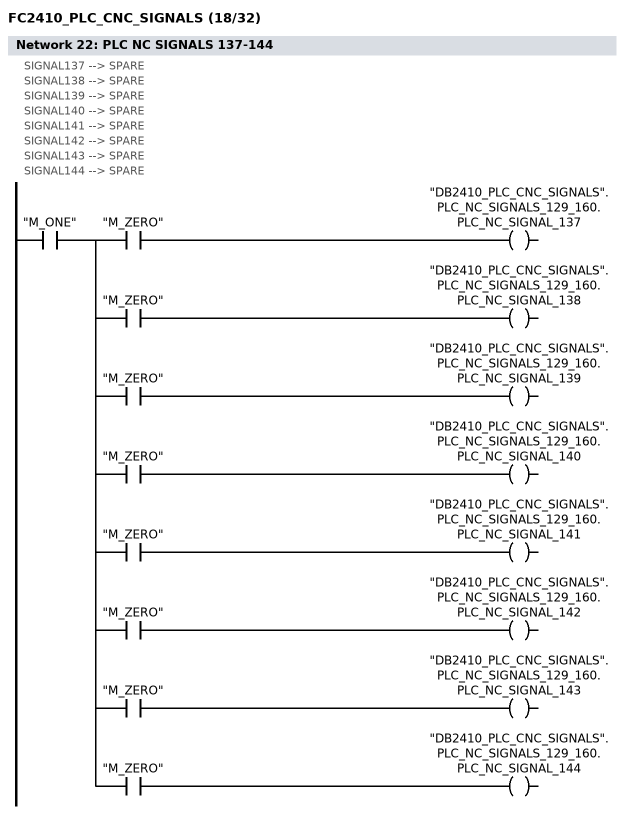
   RUNG wire#powerrail
      Contact( "M_ONE" )
      wire#w1
      Contact( "M_ZERO" )
      Coil( "DB2410_PLC_CNC_SIGNALS".PLC_NC_SIGNALS_129_160.PLC_NC_SIGNAL_137 )
   END_RUNG
   RUNG wire#w1
      Contact( "M_ZERO" )
      Coil( "DB2410_PLC_CNC_SIGNALS".PLC_NC_SIGNALS_129_160.PLC_NC_SIGNAL_138 )
   END_RUNG
   RUNG wire#w1
      Contact( "M_ZERO" )
      Coil( "DB2410_PLC_CNC_SIGNALS".PLC_NC_SIGNALS_129_160.PLC_NC_SIGNAL_139 )
   END_RUNG
   RUNG wire#w1
      Contact( "M_ZERO" )
      Coil( "DB2410_PLC_CNC_SIGNALS".PLC_NC_SIGNALS_129_160.PLC_NC_SIGNAL_140 )
   END_RUNG
   RUNG wire#w1
      Contact( "M_ZERO" )
      Coil( "DB2410_PLC_CNC_SIGNALS".PLC_NC_SIGNALS_129_160.PLC_NC_SIGNAL_141 )
   END_RUNG
   RUNG wire#w1
      Contact( "M_ZERO" )
      Coil( "DB2410_PLC_CNC_SIGNALS".PLC_NC_SIGNALS_129_160.PLC_NC_SIGNAL_142 )
   END_RUNG
   RUNG wire#w1
      Contact( "M_ZERO" )
      Coil( "DB2410_PLC_CNC_SIGNALS".PLC_NC_SIGNALS_129_160.PLC_NC_SIGNAL_143 )
   END_RUNG
   RUNG wire#w1
      Contact( "M_ZERO" )
      Coil( "DB2410_PLC_CNC_SIGNALS".PLC_NC_SIGNALS_129_160.PLC_NC_SIGNAL_144 )
   END_RUNG
   // the same network as SCL:
   "DB2410_PLC_CNC_SIGNALS".PLC_NC_SIGNALS_129_160.PLC_NC_SIGNAL_137 := "M_ONE" AND "M_ZERO";
   "DB2410_PLC_CNC_SIGNALS".PLC_NC_SIGNALS_129_160.PLC_NC_SIGNAL_138 := "M_ONE" AND "M_ZERO";
   "DB2410_PLC_CNC_SIGNALS".PLC_NC_SIGNALS_129_160.PLC_NC_SIGNAL_139 := "M_ONE" AND "M_ZERO";
   "DB2410_PLC_CNC_SIGNALS".PLC_NC_SIGNALS_129_160.PLC_NC_SIGNAL_140 := "M_ONE" AND "M_ZERO";
   "DB2410_PLC_CNC_SIGNALS".PLC_NC_SIGNALS_129_160.PLC_NC_SIGNAL_141 := "M_ONE" AND "M_ZERO";
   "DB2410_PLC_CNC_SIGNALS".PLC_NC_SIGNALS_129_160.PLC_NC_SIGNAL_142 := "M_ONE" AND "M_ZERO";
   "DB2410_PLC_CNC_SIGNALS".PLC_NC_SIGNALS_129_160.PLC_NC_SIGNAL_143 := "M_ONE" AND "M_ZERO";
   "DB2410_PLC_CNC_SIGNALS".PLC_NC_SIGNALS_129_160.PLC_NC_SIGNAL_144 := "M_ONE" AND "M_ZERO";
END_REGION

REGION Network 23: PLC NC SIGNALS 145-152
   // SIGNAL145 --> UNIT 01 FIXTURE 1 & 2 SOFTWARE ENABLED
   // SIGNAL146 --> UNIT 01 FIXTURE 3 & 4 SOFTWARE ENABLED
   // SIGNAL147 --> UNIT 02 FIXTURE 1 & 2 SOFTWARE ENABLED
   // SIGNAL148 --> UNIT 02 FIXTURE 3 & 4 SOFTWARE ENABLED
   // SIGNAL149 --> SPARE
   // SIGNAL150 --> SPARE
   // SIGNAL151 --> SPARE
   // SIGNAL152 --> SPARE
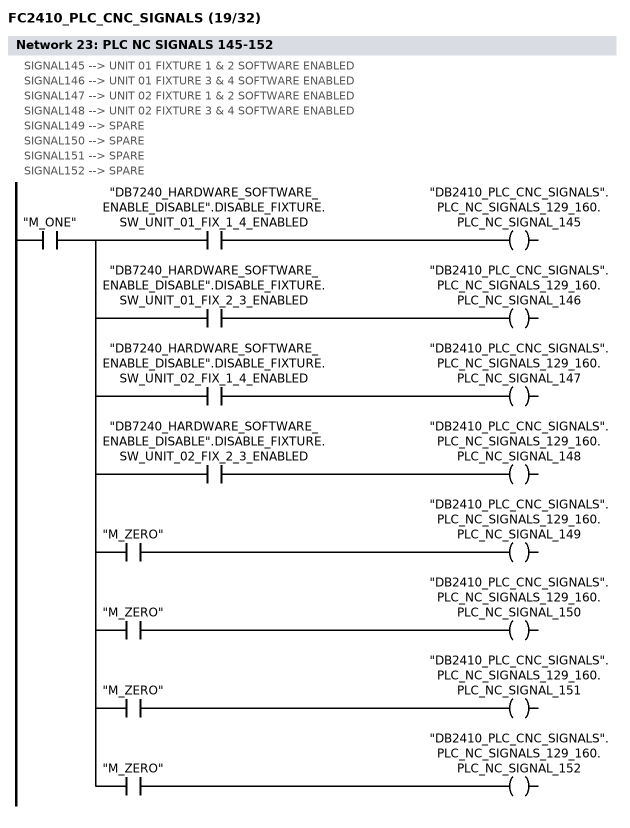
   RUNG wire#powerrail
      Contact( "M_ONE" )
      wire#w1
      Contact( "DB7240_HARDWARE_SOFTWARE_ENABLE_DISABLE".DISABLE_FIXTURE.SW_UNIT_01_FIX_1_4_ENABLED )
      Coil( "DB2410_PLC_CNC_SIGNALS".PLC_NC_SIGNALS_129_160.PLC_NC_SIGNAL_145 )
   END_RUNG
   RUNG wire#w1
      Contact( "DB7240_HARDWARE_SOFTWARE_ENABLE_DISABLE".DISABLE_FIXTURE.SW_UNIT_01_FIX_2_3_ENABLED )
      Coil( "DB2410_PLC_CNC_SIGNALS".PLC_NC_SIGNALS_129_160.PLC_NC_SIGNAL_146 )
   END_RUNG
   RUNG wire#w1
      Contact( "DB7240_HARDWARE_SOFTWARE_ENABLE_DISABLE".DISABLE_FIXTURE.SW_UNIT_02_FIX_1_4_ENABLED )
      Coil( "DB2410_PLC_CNC_SIGNALS".PLC_NC_SIGNALS_129_160.PLC_NC_SIGNAL_147 )
   END_RUNG
   RUNG wire#w1
      Contact( "DB7240_HARDWARE_SOFTWARE_ENABLE_DISABLE".DISABLE_FIXTURE.SW_UNIT_02_FIX_2_3_ENABLED )
      Coil( "DB2410_PLC_CNC_SIGNALS".PLC_NC_SIGNALS_129_160.PLC_NC_SIGNAL_148 )
   END_RUNG
   RUNG wire#w1
      Contact( "M_ZERO" )
      Coil( "DB2410_PLC_CNC_SIGNALS".PLC_NC_SIGNALS_129_160.PLC_NC_SIGNAL_149 )
   END_RUNG
   RUNG wire#w1
      Contact( "M_ZERO" )
      Coil( "DB2410_PLC_CNC_SIGNALS".PLC_NC_SIGNALS_129_160.PLC_NC_SIGNAL_150 )
   END_RUNG
   RUNG wire#w1
      Contact( "M_ZERO" )
      Coil( "DB2410_PLC_CNC_SIGNALS".PLC_NC_SIGNALS_129_160.PLC_NC_SIGNAL_151 )
   END_RUNG
   RUNG wire#w1
      Contact( "M_ZERO" )
      Coil( "DB2410_PLC_CNC_SIGNALS".PLC_NC_SIGNALS_129_160.PLC_NC_SIGNAL_152 )
   END_RUNG
   // the same network as SCL:
   "DB2410_PLC_CNC_SIGNALS".PLC_NC_SIGNALS_129_160.PLC_NC_SIGNAL_145 := "M_ONE" AND "DB7240_HARDWARE_SOFTWARE_ENABLE_DISABLE".DISABLE_FIXTURE.SW_UNIT_01_FIX_1_4_ENABLED;
   "DB2410_PLC_CNC_SIGNALS".PLC_NC_SIGNALS_129_160.PLC_NC_SIGNAL_146 := "M_ONE" AND "DB7240_HARDWARE_SOFTWARE_ENABLE_DISABLE".DISABLE_FIXTURE.SW_UNIT_01_FIX_2_3_ENABLED;
   "DB2410_PLC_CNC_SIGNALS".PLC_NC_SIGNALS_129_160.PLC_NC_SIGNAL_147 := "M_ONE" AND "DB7240_HARDWARE_SOFTWARE_ENABLE_DISABLE".DISABLE_FIXTURE.SW_UNIT_02_FIX_1_4_ENABLED;
   "DB2410_PLC_CNC_SIGNALS".PLC_NC_SIGNALS_129_160.PLC_NC_SIGNAL_148 := "M_ONE" AND "DB7240_HARDWARE_SOFTWARE_ENABLE_DISABLE".DISABLE_FIXTURE.SW_UNIT_02_FIX_2_3_ENABLED;
   "DB2410_PLC_CNC_SIGNALS".PLC_NC_SIGNALS_129_160.PLC_NC_SIGNAL_149 := "M_ONE" AND "M_ZERO";
   "DB2410_PLC_CNC_SIGNALS".PLC_NC_SIGNALS_129_160.PLC_NC_SIGNAL_150 := "M_ONE" AND "M_ZERO";
   "DB2410_PLC_CNC_SIGNALS".PLC_NC_SIGNALS_129_160.PLC_NC_SIGNAL_151 := "M_ONE" AND "M_ZERO";
   "DB2410_PLC_CNC_SIGNALS".PLC_NC_SIGNALS_129_160.PLC_NC_SIGNAL_152 := "M_ONE" AND "M_ZERO";
END_REGION

REGION Network 24: PLC NC SIGNALS 153-160
   // SIGNAL153 --> SPARE
   // SIGNAL154 --> SPARE
   // SIGNAL155 --> SPARE
   // SIGNAL156 --> SPARE
   // SIGNAL157 --> SPARE
   // SIGNAL158 --> SPARE
   // SIGNAL159 --> SPARE
   // SIGNAL160 --> SPARE
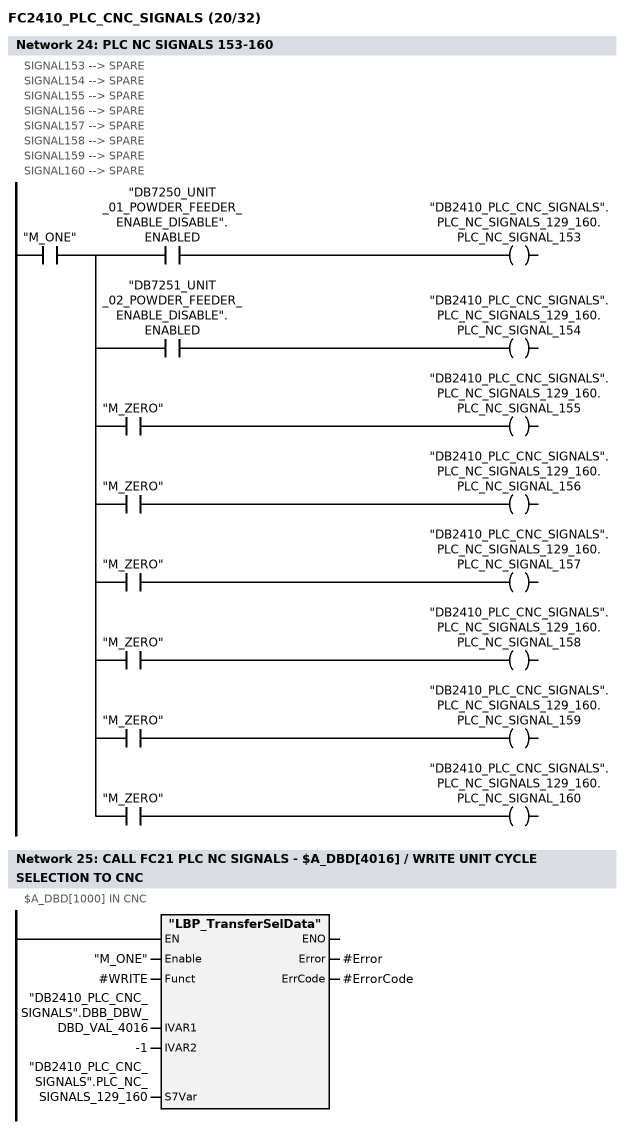
   RUNG wire#powerrail
      Contact( "M_ONE" )
      wire#w1
      Contact( "DB7250_UNIT _01_POWDER_FEEDER_ENABLE_DISABLE".ENABLED )
      Coil( "DB2410_PLC_CNC_SIGNALS".PLC_NC_SIGNALS_129_160.PLC_NC_SIGNAL_153 )
   END_RUNG
   RUNG wire#w1
      Contact( "DB7251_UNIT _02_POWDER_FEEDER_ENABLE_DISABLE".ENABLED )
      Coil( "DB2410_PLC_CNC_SIGNALS".PLC_NC_SIGNALS_129_160.PLC_NC_SIGNAL_154 )
   END_RUNG
   RUNG wire#w1
      Contact( "M_ZERO" )
      Coil( "DB2410_PLC_CNC_SIGNALS".PLC_NC_SIGNALS_129_160.PLC_NC_SIGNAL_155 )
   END_RUNG
   RUNG wire#w1
      Contact( "M_ZERO" )
      Coil( "DB2410_PLC_CNC_SIGNALS".PLC_NC_SIGNALS_129_160.PLC_NC_SIGNAL_156 )
   END_RUNG
   RUNG wire#w1
      Contact( "M_ZERO" )
      Coil( "DB2410_PLC_CNC_SIGNALS".PLC_NC_SIGNALS_129_160.PLC_NC_SIGNAL_157 )
   END_RUNG
   RUNG wire#w1
      Contact( "M_ZERO" )
      Coil( "DB2410_PLC_CNC_SIGNALS".PLC_NC_SIGNALS_129_160.PLC_NC_SIGNAL_158 )
   END_RUNG
   RUNG wire#w1
      Contact( "M_ZERO" )
      Coil( "DB2410_PLC_CNC_SIGNALS".PLC_NC_SIGNALS_129_160.PLC_NC_SIGNAL_159 )
   END_RUNG
   RUNG wire#w1
      Contact( "M_ZERO" )
      Coil( "DB2410_PLC_CNC_SIGNALS".PLC_NC_SIGNALS_129_160.PLC_NC_SIGNAL_160 )
   END_RUNG
   // the same network as SCL:
   "DB2410_PLC_CNC_SIGNALS".PLC_NC_SIGNALS_129_160.PLC_NC_SIGNAL_153 := "M_ONE" AND "DB7250_UNIT _01_POWDER_FEEDER_ENABLE_DISABLE".ENABLED;
   "DB2410_PLC_CNC_SIGNALS".PLC_NC_SIGNALS_129_160.PLC_NC_SIGNAL_154 := "M_ONE" AND "DB7251_UNIT _02_POWDER_FEEDER_ENABLE_DISABLE".ENABLED;
   "DB2410_PLC_CNC_SIGNALS".PLC_NC_SIGNALS_129_160.PLC_NC_SIGNAL_155 := "M_ONE" AND "M_ZERO";
   "DB2410_PLC_CNC_SIGNALS".PLC_NC_SIGNALS_129_160.PLC_NC_SIGNAL_156 := "M_ONE" AND "M_ZERO";
   "DB2410_PLC_CNC_SIGNALS".PLC_NC_SIGNALS_129_160.PLC_NC_SIGNAL_157 := "M_ONE" AND "M_ZERO";
   "DB2410_PLC_CNC_SIGNALS".PLC_NC_SIGNALS_129_160.PLC_NC_SIGNAL_158 := "M_ONE" AND "M_ZERO";
   "DB2410_PLC_CNC_SIGNALS".PLC_NC_SIGNALS_129_160.PLC_NC_SIGNAL_159 := "M_ONE" AND "M_ZERO";
   "DB2410_PLC_CNC_SIGNALS".PLC_NC_SIGNALS_129_160.PLC_NC_SIGNAL_160 := "M_ONE" AND "M_ZERO";
END_REGION

REGION Network 25: CALL FC21 PLC NC SIGNALS - $A_DBD[4016] / WRITE UNIT CYCLE SELECTION TO CNC
   // $A_DBD[1000] IN CNC
   RUNG wire#powerrail
      "LBP_TransferSelData"(Enable := "M_ONE", Funct := #WRITE, IVAR1 := "DB2410_PLC_CNC_SIGNALS".DBB_DBW_DBD_VAL_4016, IVAR2 := -1, S7Var := "DB2410_PLC_CNC_SIGNALS".PLC_NC_SIGNALS_129_160, Error => #Error, ErrCode => #ErrorCode)
   END_RUNG
   // the same network as SCL:
   "LBP_TransferSelData"(Enable := "M_ONE",
                         Funct := #WRITE,
                         IVAR1 := "DB2410_PLC_CNC_SIGNALS".DBB_DBW_DBD_VAL_4016,
                         IVAR2 := -1,
                         S7Var := "DB2410_PLC_CNC_SIGNALS".PLC_NC_SIGNALS_129_160,
                         Error => #Error,
                         ErrCode => #ErrorCode);
END_REGION

REGION Network 26: PLC NC SIGNALS 161-168
   // SIGNAL161 --> BK MIKRO SP11 ENABLED
   // SIGNAL162 --> BK MIKRO SP12 ENABLED
   // SIGNAL163 --> BK MIKRO SP13 ENABLED
   // SIGNAL164 --> BK MIKRO SP14 ENABLED
   // SIGNAL165 --> SPARE
   // SIGNAL166 --> SPARE
   // SIGNAL167 --> SPARE
   // SIGNAL168 --> SPARE
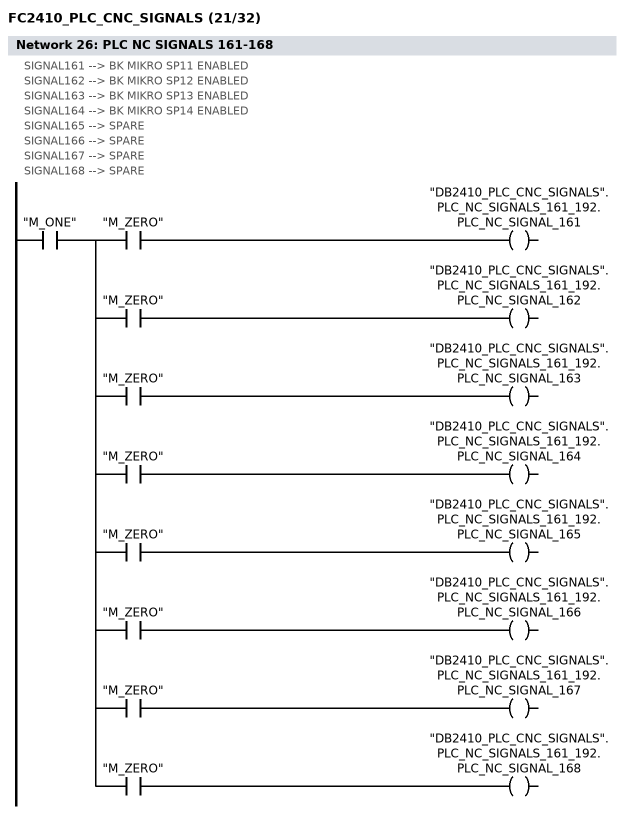
   RUNG wire#powerrail
      Contact( "M_ONE" )
      wire#w1
      Contact( "M_ZERO" )
      Coil( "DB2410_PLC_CNC_SIGNALS".PLC_NC_SIGNALS_161_192.PLC_NC_SIGNAL_161 )
   END_RUNG
   RUNG wire#w1
      Contact( "M_ZERO" )
      Coil( "DB2410_PLC_CNC_SIGNALS".PLC_NC_SIGNALS_161_192.PLC_NC_SIGNAL_162 )
   END_RUNG
   RUNG wire#w1
      Contact( "M_ZERO" )
      Coil( "DB2410_PLC_CNC_SIGNALS".PLC_NC_SIGNALS_161_192.PLC_NC_SIGNAL_163 )
   END_RUNG
   RUNG wire#w1
      Contact( "M_ZERO" )
      Coil( "DB2410_PLC_CNC_SIGNALS".PLC_NC_SIGNALS_161_192.PLC_NC_SIGNAL_164 )
   END_RUNG
   RUNG wire#w1
      Contact( "M_ZERO" )
      Coil( "DB2410_PLC_CNC_SIGNALS".PLC_NC_SIGNALS_161_192.PLC_NC_SIGNAL_165 )
   END_RUNG
   RUNG wire#w1
      Contact( "M_ZERO" )
      Coil( "DB2410_PLC_CNC_SIGNALS".PLC_NC_SIGNALS_161_192.PLC_NC_SIGNAL_166 )
   END_RUNG
   RUNG wire#w1
      Contact( "M_ZERO" )
      Coil( "DB2410_PLC_CNC_SIGNALS".PLC_NC_SIGNALS_161_192.PLC_NC_SIGNAL_167 )
   END_RUNG
   RUNG wire#w1
      Contact( "M_ZERO" )
      Coil( "DB2410_PLC_CNC_SIGNALS".PLC_NC_SIGNALS_161_192.PLC_NC_SIGNAL_168 )
   END_RUNG
   // the same network as SCL:
   "DB2410_PLC_CNC_SIGNALS".PLC_NC_SIGNALS_161_192.PLC_NC_SIGNAL_161 := "M_ONE" AND "M_ZERO";
   "DB2410_PLC_CNC_SIGNALS".PLC_NC_SIGNALS_161_192.PLC_NC_SIGNAL_162 := "M_ONE" AND "M_ZERO";
   "DB2410_PLC_CNC_SIGNALS".PLC_NC_SIGNALS_161_192.PLC_NC_SIGNAL_163 := "M_ONE" AND "M_ZERO";
   "DB2410_PLC_CNC_SIGNALS".PLC_NC_SIGNALS_161_192.PLC_NC_SIGNAL_164 := "M_ONE" AND "M_ZERO";
   "DB2410_PLC_CNC_SIGNALS".PLC_NC_SIGNALS_161_192.PLC_NC_SIGNAL_165 := "M_ONE" AND "M_ZERO";
   "DB2410_PLC_CNC_SIGNALS".PLC_NC_SIGNALS_161_192.PLC_NC_SIGNAL_166 := "M_ONE" AND "M_ZERO";
   "DB2410_PLC_CNC_SIGNALS".PLC_NC_SIGNALS_161_192.PLC_NC_SIGNAL_167 := "M_ONE" AND "M_ZERO";
   "DB2410_PLC_CNC_SIGNALS".PLC_NC_SIGNALS_161_192.PLC_NC_SIGNAL_168 := "M_ONE" AND "M_ZERO";
END_REGION

REGION Network 27: PLC NC SIGNALS 169-176
   // SIGNAL169 --> BK MIKRO SP21 ENABLED
   // SIGNAL170 --> BK MIKRO SP22 ENABLED
   // SIGNAL171 --> BK MIKRO SP23 ENABLED
   // SIGNAL172 --> BK MIKRO SP24 ENABLED
   // SIGNAL173 --> SPARE
   // SIGNAL174 --> SPARE
   // SIGNAL175 --> SPARE
   // SIGNAL176 --> SPARE
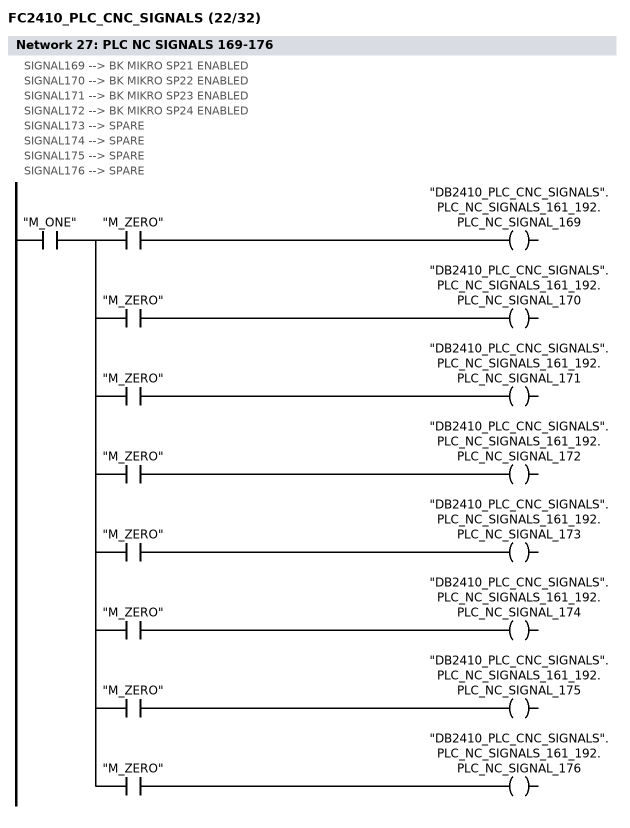
   RUNG wire#powerrail
      Contact( "M_ONE" )
      wire#w1
      Contact( "M_ZERO" )
      Coil( "DB2410_PLC_CNC_SIGNALS".PLC_NC_SIGNALS_161_192.PLC_NC_SIGNAL_169 )
   END_RUNG
   RUNG wire#w1
      Contact( "M_ZERO" )
      Coil( "DB2410_PLC_CNC_SIGNALS".PLC_NC_SIGNALS_161_192.PLC_NC_SIGNAL_170 )
   END_RUNG
   RUNG wire#w1
      Contact( "M_ZERO" )
      Coil( "DB2410_PLC_CNC_SIGNALS".PLC_NC_SIGNALS_161_192.PLC_NC_SIGNAL_171 )
   END_RUNG
   RUNG wire#w1
      Contact( "M_ZERO" )
      Coil( "DB2410_PLC_CNC_SIGNALS".PLC_NC_SIGNALS_161_192.PLC_NC_SIGNAL_172 )
   END_RUNG
   RUNG wire#w1
      Contact( "M_ZERO" )
      Coil( "DB2410_PLC_CNC_SIGNALS".PLC_NC_SIGNALS_161_192.PLC_NC_SIGNAL_173 )
   END_RUNG
   RUNG wire#w1
      Contact( "M_ZERO" )
      Coil( "DB2410_PLC_CNC_SIGNALS".PLC_NC_SIGNALS_161_192.PLC_NC_SIGNAL_174 )
   END_RUNG
   RUNG wire#w1
      Contact( "M_ZERO" )
      Coil( "DB2410_PLC_CNC_SIGNALS".PLC_NC_SIGNALS_161_192.PLC_NC_SIGNAL_175 )
   END_RUNG
   RUNG wire#w1
      Contact( "M_ZERO" )
      Coil( "DB2410_PLC_CNC_SIGNALS".PLC_NC_SIGNALS_161_192.PLC_NC_SIGNAL_176 )
   END_RUNG
   // the same network as SCL:
   "DB2410_PLC_CNC_SIGNALS".PLC_NC_SIGNALS_161_192.PLC_NC_SIGNAL_169 := "M_ONE" AND "M_ZERO";
   "DB2410_PLC_CNC_SIGNALS".PLC_NC_SIGNALS_161_192.PLC_NC_SIGNAL_170 := "M_ONE" AND "M_ZERO";
   "DB2410_PLC_CNC_SIGNALS".PLC_NC_SIGNALS_161_192.PLC_NC_SIGNAL_171 := "M_ONE" AND "M_ZERO";
   "DB2410_PLC_CNC_SIGNALS".PLC_NC_SIGNALS_161_192.PLC_NC_SIGNAL_172 := "M_ONE" AND "M_ZERO";
   "DB2410_PLC_CNC_SIGNALS".PLC_NC_SIGNALS_161_192.PLC_NC_SIGNAL_173 := "M_ONE" AND "M_ZERO";
   "DB2410_PLC_CNC_SIGNALS".PLC_NC_SIGNALS_161_192.PLC_NC_SIGNAL_174 := "M_ONE" AND "M_ZERO";
   "DB2410_PLC_CNC_SIGNALS".PLC_NC_SIGNALS_161_192.PLC_NC_SIGNAL_175 := "M_ONE" AND "M_ZERO";
   "DB2410_PLC_CNC_SIGNALS".PLC_NC_SIGNALS_161_192.PLC_NC_SIGNAL_176 := "M_ONE" AND "M_ZERO";
END_REGION

REGION Network 28: PLC NC SIGNALS 177-184
   // SIGNAL177 --> BK MIKRO TOOL BREAKAGE 01R
   // SIGNAL178 --> BK MIKRO SP11 BROKEN
   // SIGNAL179 --> BK MIKRO SP12 BROKEN
   // SIGNAL180 --> BK MIKRO SP13 BROKEN
   // SIGNAL181 --> BK MIKRO SP14 BROKEN
   // SIGNAL182 --> SPARE
   // SIGNAL183 --> SPARE
   // SIGNAL184 --> SPARE
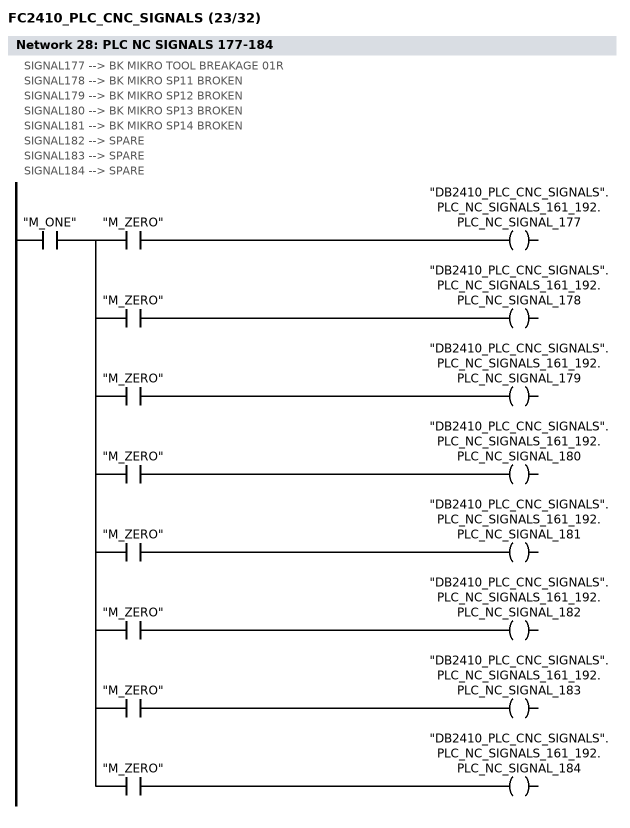
   RUNG wire#powerrail
      Contact( "M_ONE" )
      wire#w1
      Contact( "M_ZERO" )
      Coil( "DB2410_PLC_CNC_SIGNALS".PLC_NC_SIGNALS_161_192.PLC_NC_SIGNAL_177 )
   END_RUNG
   RUNG wire#w1
      Contact( "M_ZERO" )
      Coil( "DB2410_PLC_CNC_SIGNALS".PLC_NC_SIGNALS_161_192.PLC_NC_SIGNAL_178 )
   END_RUNG
   RUNG wire#w1
      Contact( "M_ZERO" )
      Coil( "DB2410_PLC_CNC_SIGNALS".PLC_NC_SIGNALS_161_192.PLC_NC_SIGNAL_179 )
   END_RUNG
   RUNG wire#w1
      Contact( "M_ZERO" )
      Coil( "DB2410_PLC_CNC_SIGNALS".PLC_NC_SIGNALS_161_192.PLC_NC_SIGNAL_180 )
   END_RUNG
   RUNG wire#w1
      Contact( "M_ZERO" )
      Coil( "DB2410_PLC_CNC_SIGNALS".PLC_NC_SIGNALS_161_192.PLC_NC_SIGNAL_181 )
   END_RUNG
   RUNG wire#w1
      Contact( "M_ZERO" )
      Coil( "DB2410_PLC_CNC_SIGNALS".PLC_NC_SIGNALS_161_192.PLC_NC_SIGNAL_182 )
   END_RUNG
   RUNG wire#w1
      Contact( "M_ZERO" )
      Coil( "DB2410_PLC_CNC_SIGNALS".PLC_NC_SIGNALS_161_192.PLC_NC_SIGNAL_183 )
   END_RUNG
   RUNG wire#w1
      Contact( "M_ZERO" )
      Coil( "DB2410_PLC_CNC_SIGNALS".PLC_NC_SIGNALS_161_192.PLC_NC_SIGNAL_184 )
   END_RUNG
   // the same network as SCL:
   "DB2410_PLC_CNC_SIGNALS".PLC_NC_SIGNALS_161_192.PLC_NC_SIGNAL_177 := "M_ONE" AND "M_ZERO";
   "DB2410_PLC_CNC_SIGNALS".PLC_NC_SIGNALS_161_192.PLC_NC_SIGNAL_178 := "M_ONE" AND "M_ZERO";
   "DB2410_PLC_CNC_SIGNALS".PLC_NC_SIGNALS_161_192.PLC_NC_SIGNAL_179 := "M_ONE" AND "M_ZERO";
   "DB2410_PLC_CNC_SIGNALS".PLC_NC_SIGNALS_161_192.PLC_NC_SIGNAL_180 := "M_ONE" AND "M_ZERO";
   "DB2410_PLC_CNC_SIGNALS".PLC_NC_SIGNALS_161_192.PLC_NC_SIGNAL_181 := "M_ONE" AND "M_ZERO";
   "DB2410_PLC_CNC_SIGNALS".PLC_NC_SIGNALS_161_192.PLC_NC_SIGNAL_182 := "M_ONE" AND "M_ZERO";
   "DB2410_PLC_CNC_SIGNALS".PLC_NC_SIGNALS_161_192.PLC_NC_SIGNAL_183 := "M_ONE" AND "M_ZERO";
   "DB2410_PLC_CNC_SIGNALS".PLC_NC_SIGNALS_161_192.PLC_NC_SIGNAL_184 := "M_ONE" AND "M_ZERO";
END_REGION

REGION Network 29: PLC NC SIGNALS 185-192
   // SIGNAL185 --> BK MIKRO TOOL BREAKAGE 01L
   // SIGNAL186 --> BK MIKRO SP21 BROKEN
   // SIGNAL187 --> BK MIKRO SP22 BROKEN
   // SIGNAL188 --> BK MIKRO SP23 BROKEN
   // SIGNAL189 --> BK MIKRO SP24 BROKEN
   // SIGNAL190 --> SPARE
   // SIGNAL191 --> SPARE
   // SIGNAL192 --> SPARE
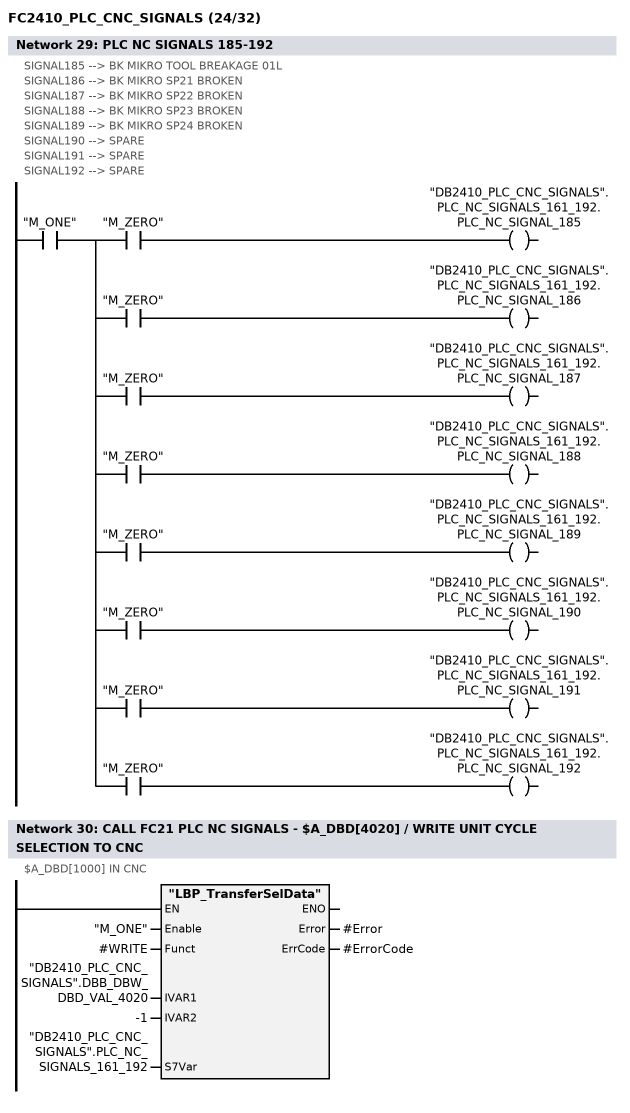
   RUNG wire#powerrail
      Contact( "M_ONE" )
      wire#w1
      Contact( "M_ZERO" )
      Coil( "DB2410_PLC_CNC_SIGNALS".PLC_NC_SIGNALS_161_192.PLC_NC_SIGNAL_185 )
   END_RUNG
   RUNG wire#w1
      Contact( "M_ZERO" )
      Coil( "DB2410_PLC_CNC_SIGNALS".PLC_NC_SIGNALS_161_192.PLC_NC_SIGNAL_186 )
   END_RUNG
   RUNG wire#w1
      Contact( "M_ZERO" )
      Coil( "DB2410_PLC_CNC_SIGNALS".PLC_NC_SIGNALS_161_192.PLC_NC_SIGNAL_187 )
   END_RUNG
   RUNG wire#w1
      Contact( "M_ZERO" )
      Coil( "DB2410_PLC_CNC_SIGNALS".PLC_NC_SIGNALS_161_192.PLC_NC_SIGNAL_188 )
   END_RUNG
   RUNG wire#w1
      Contact( "M_ZERO" )
      Coil( "DB2410_PLC_CNC_SIGNALS".PLC_NC_SIGNALS_161_192.PLC_NC_SIGNAL_189 )
   END_RUNG
   RUNG wire#w1
      Contact( "M_ZERO" )
      Coil( "DB2410_PLC_CNC_SIGNALS".PLC_NC_SIGNALS_161_192.PLC_NC_SIGNAL_190 )
   END_RUNG
   RUNG wire#w1
      Contact( "M_ZERO" )
      Coil( "DB2410_PLC_CNC_SIGNALS".PLC_NC_SIGNALS_161_192.PLC_NC_SIGNAL_191 )
   END_RUNG
   RUNG wire#w1
      Contact( "M_ZERO" )
      Coil( "DB2410_PLC_CNC_SIGNALS".PLC_NC_SIGNALS_161_192.PLC_NC_SIGNAL_192 )
   END_RUNG
   // the same network as SCL:
   "DB2410_PLC_CNC_SIGNALS".PLC_NC_SIGNALS_161_192.PLC_NC_SIGNAL_185 := "M_ONE" AND "M_ZERO";
   "DB2410_PLC_CNC_SIGNALS".PLC_NC_SIGNALS_161_192.PLC_NC_SIGNAL_186 := "M_ONE" AND "M_ZERO";
   "DB2410_PLC_CNC_SIGNALS".PLC_NC_SIGNALS_161_192.PLC_NC_SIGNAL_187 := "M_ONE" AND "M_ZERO";
   "DB2410_PLC_CNC_SIGNALS".PLC_NC_SIGNALS_161_192.PLC_NC_SIGNAL_188 := "M_ONE" AND "M_ZERO";
   "DB2410_PLC_CNC_SIGNALS".PLC_NC_SIGNALS_161_192.PLC_NC_SIGNAL_189 := "M_ONE" AND "M_ZERO";
   "DB2410_PLC_CNC_SIGNALS".PLC_NC_SIGNALS_161_192.PLC_NC_SIGNAL_190 := "M_ONE" AND "M_ZERO";
   "DB2410_PLC_CNC_SIGNALS".PLC_NC_SIGNALS_161_192.PLC_NC_SIGNAL_191 := "M_ONE" AND "M_ZERO";
   "DB2410_PLC_CNC_SIGNALS".PLC_NC_SIGNALS_161_192.PLC_NC_SIGNAL_192 := "M_ONE" AND "M_ZERO";
END_REGION

REGION Network 30: CALL FC21 PLC NC SIGNALS - $A_DBD[4020] / WRITE UNIT CYCLE SELECTION TO CNC
   // $A_DBD[1000] IN CNC
   RUNG wire#powerrail
      "LBP_TransferSelData"(Enable := "M_ONE", Funct := #WRITE, IVAR1 := "DB2410_PLC_CNC_SIGNALS".DBB_DBW_DBD_VAL_4020, IVAR2 := -1, S7Var := "DB2410_PLC_CNC_SIGNALS".PLC_NC_SIGNALS_161_192, Error => #Error, ErrCode => #ErrorCode)
   END_RUNG
   // the same network as SCL:
   "LBP_TransferSelData"(Enable := "M_ONE",
                         Funct := #WRITE,
                         IVAR1 := "DB2410_PLC_CNC_SIGNALS".DBB_DBW_DBD_VAL_4020,
                         IVAR2 := -1,
                         S7Var := "DB2410_PLC_CNC_SIGNALS".PLC_NC_SIGNALS_161_192,
                         Error => #Error,
                         ErrCode => #ErrorCode);
END_REGION

REGION Network 31: PLC NC SIGNALS 193-200
   // SIGNAL193 --> PROBE ENABLED PART A
   // SIGNAL194 --> PROBE ENABLED PART B
   // SIGNAL195 --> PROBE ENABLED PART C
   // SIGNAL196 --> SPARE
   // SIGNAL197 --> SPARE
   // SIGNAL198 --> SPARE
   // SIGNAL199 --> SPARE
   // SIGNAL200 --> SPARE
